KUKA KRL program: MyProgram_238().src

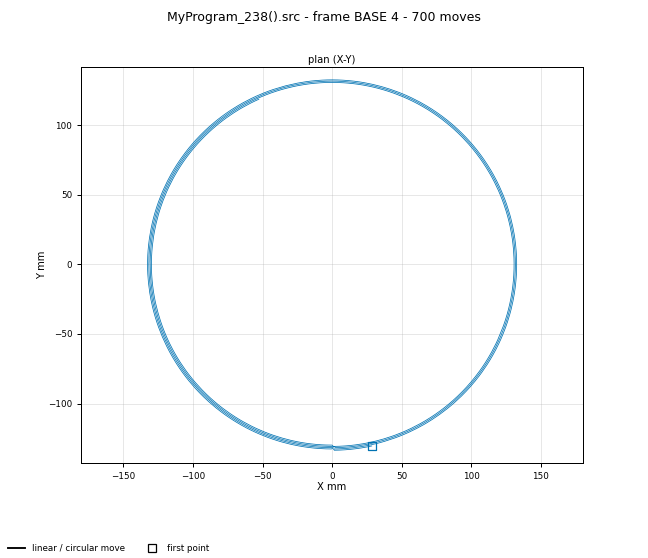
[picture p0: tool path of MyProgram_238().src in frame BASE 4, 700 of 700 moves have a stored position in this frame; points joined in program order, loops and branches not executed]
&ACCESS RVP
&REL 1
&PARAM TEMPLATE = C:\KRC\Roboter\Template\vorgabe
&PARAM EDITMASK = *
DEF MyProgram_238()
; ---- Setting reference (Base) ----
$BASE = BASE_DATA[4]

; --------------------------
; ---- Setting tool (TCP) ----
$TOOL = TOOL_DATA[3]
; --------------------------

$VEL.CP = VEL_APROX_PRINT
Startdeposition()
$VEL.CP = VEL_PRINT
LIN {X 28.5012,Y -130.5198,Z 160,A -79.1716,B 19.6548,C -0.4337,E1 19.6933,E2 527.426} C_DIS
LIN {X 25.4461,Y -131.1499,Z 160,A -80.7496,B 19.6549,C -0.4225,E1 19.6889,E2 529.0345} C_DIS
LIN {X 21.1826,Y -131.9073,Z 160,A -82.61,B 19.6549,C -0.4211,E1 19.6838,E2 530.8968} C_DIS
LIN {X 17.506,Y -132.4434,Z 160,A -84.1425,B 19.6549,C -0.4226,E1 19.6796,E2 532.4228} C_DIS
LIN {X 13.4148,Y -132.9217,Z 160,A -85.958,B 19.6549,C -0.4196,E1 19.6745,E2 534.2456} C_DIS
LIN {X 9.6729,Y -133.2447,Z 160,A -87.4931,B 19.6549,C -0.4221,E1 19.6703,E2 535.7723} C_DIS
LIN {X 5.6097,Y -133.4781,Z 160,A -89.2555,B 19.6549,C -0.4208,E1 19.6653,E2 537.5378} C_DIS
LIN {X 1.5658,Y -133.5878,Z 160,A -91.031,B 19.655,C -0.4187,E1 19.6604,E2 539.3193} C_DIS
LIN {X 1.5658,Y -133.5878,Z 160,A -91.031,B 19.655,C -0.4187,E1 19.6604,E2 539.3193} C_DIS
Enddeposition()
LIN {X 0.9434,Y -132.6616,Z 160,A -90.6102,B 18.4313,C -0.2923,E1 18.435,E2 539.1863} C_DIS
Startdeposition()
$VEL.CP = VEL_PRINT
LIN {X 3.7021,Y -132.6178,Z 160,A -88.9683,B 18.4311,C -0.31,E1 18.4397,E2 537.489} C_DIS
LIN {X 7.8936,Y -132.4346,Z 160,A -87.1638,B 18.4311,C -0.3103,E1 18.4447,E2 535.6844} C_DIS
LIN {X 11.5593,Y -132.1654,Z 160,A -85.513,B 18.431,C -0.3135,E1 18.4494,E2 534.0249} C_DIS
LIN {X 15.642,Y -131.744,Z 160,A -83.8719,B 18.431,C -0.3092,E1 18.4539,E2 532.3987} C_DIS
LIN {X 18.8772,Y -131.3195,Z 160,A -82.4668,B 18.431,C -0.3099,E1 18.4578,E2 530.9931} C_DIS
LIN {X 22.0168,Y -130.8298,Z 160,A -81.0377,B 18.431,C -0.3131,E1 18.4617,E2 529.556} C_DIS
LIN {X 27.2844,Y -129.8353,Z 160,A -78.6667,B 18.431,C -0.3171,E1 18.4682,E2 527.1765} C_DIS
LIN {X 31.009,Y -128.9944,Z 160,A -77.1259,B 18.431,C -0.3143,E1 18.4724,E2 525.6476} C_DIS
LIN {X 34.2185,Y -128.1803,Z 160,A -75.6772,B 18.431,C -0.3164,E1 18.4763,E2 524.1953} C_DIS
LIN {X 37.7119,Y -127.1971,Z 160,A -73.4165,B 18.4304,C -0.3458,E1 18.4826,E2 521.8475} C_DIS
LIN {X 42.8714,Y -125.5528,Z 160,A -71.8794,B 18.4309,C -0.3163,E1 18.4864,E2 520.4075} C_DIS
LIN {X 45.287,Y -124.7006,Z 160,A -70.7303,B 18.4309,C -0.3194,E1 18.4895,E2 519.2521} C_DIS
LIN {X 48.16,Y -123.6191,Z 160,A -69.3935,B 18.4309,C -0.3215,E1 18.493,E2 517.9126} C_DIS
LIN {X 51.5502,Y -122.245,Z 160,A -67.7549,B 18.4308,C -0.326,E1 18.4972,E2 516.2652} C_DIS
LIN {X 55.221,Y -120.6314,Z 160,A -65.2452,B 18.4302,C -0.36,E1 18.5038,E2 513.6571} C_DIS
LIN {X 60.6173,Y -118.0119,Z 160,A -63.7627,B 18.4309,C -0.3191,E1 18.5072,E2 512.3091} C_DIS
LIN {X 65.5426,Y -115.3507,Z 160,A -61.2737,B 18.4308,C -0.3259,E1 18.5133,E2 509.8088} C_DIS
LIN {X 68.1939,Y -113.8036,Z 160,A -59.6762,B 18.4306,C -0.3392,E1 18.5173,E2 508.1764} C_DIS
LIN {X 71.8599,Y -111.5251,Z 160,A -56.9687,B 18.4298,C -0.3771,E1 18.5239,E2 505.3617} C_DIS
LIN {X 77.3198,Y -107.8111,Z 160,A -55.0523,B 18.4305,C -0.3442,E1 18.528,E2 503.5582} C_DIS
LIN {X 82.5623,Y -103.851,Z 160,A -52.1665,B 18.4303,C -0.3519,E1 18.5344,E2 500.6629} C_DIS
LIN {X 85.006,Y -101.861,Z 160,A -50.9012,B 18.4303,C -0.3509,E1 18.5371,E2 499.4076} C_DIS
LIN {X 87.8381,Y -99.4285,Z 160,A -49.2007,B 18.4303,C -0.358,E1 18.5407,E2 497.6941} C_DIS
LIN {X 92.702,Y -94.91,Z 160,A -46.2129,B 18.43,C -0.3695,E1 18.5468,E2 494.6876} C_DIS
LIN {X 96.1781,Y -91.3865,Z 160,A -44.2202,B 18.43,C -0.3685,E1 18.5506,E2 492.7098} C_DIS
LIN {X 99.1469,Y -88.1567,Z 160,A -41.7561,B 18.4294,C -0.3968,E1 18.5554,E2 490.1723} C_DIS
LIN {X 102.5594,Y -84.1613,Z 160,A -40.2554,B 18.43,C -0.3705,E1 18.5579,E2 488.7637} C_DIS
LIN {X 105.6485,Y -80.2491,Z 160,A -37.9278,B 18.4297,C -0.3833,E1 18.5619,E2 486.4115} C_DIS
LIN {X 107.5535,Y -77.6779,Z 160,A -36.4631,B 18.4296,C -0.3903,E1 18.5643,E2 484.9345} C_DIS
LIN {X 111.3907,Y -72.0675,Z 160,A -33.8423,B 18.4296,C -0.3851,E1 18.5684,E2 482.3483} C_DIS
LIN {X 113.2763,Y -69.0665,Z 160,A -32.1365,B 18.4295,C -0.3965,E1 18.5709,E2 480.6186} C_DIS
LIN {X 115.4572,Y -65.3557,Z 160,A -30.138,B 18.4292,C -0.4075,E1 18.5737,E2 478.6} C_DIS
LIN {X 117.6562,Y -61.3044,Z 160,A -28.4402,B 18.4294,C -0.401,E1 18.5759,E2 476.9354} C_DIS
LIN {X 119.8553,Y -56.8847,Z 160,A -26.3011,B 18.4292,C -0.4074,E1 18.5785,E2 474.7922} C_DIS
LIN {X 121.3634,Y -53.5945,Z 160,A -24.7471,B 18.4292,C -0.4115,E1 18.5803,E2 473.2369} C_DIS
LIN {X 122.9377,Y -49.8746,Z 160,A -22.4308,B 18.4285,C -0.4406,E1 18.5828,E2 470.8472} C_DIS
LIN {X 124.6788,Y -45.3476,Z 160,A -21.1339,B 18.4291,C -0.4134,E1 18.584,E2 469.6456} C_DIS
LIN {X 126.0019,Y -41.5302,Z 160,A -19.0898,B 18.4287,C -0.4311,E1 18.5858,E2 467.5621} C_DIS
LIN {X 127.7829,Y -35.6739,Z 160,A -16.6066,B 18.4287,C -0.4324,E1 18.5878,E2 465.0946} C_DIS
LIN {X 128.6356,Y -32.4655,Z 160,A -15.1512,B 18.4286,C -0.4377,E1 18.5888,E2 463.6344} C_DIS
LIN {X 130.0281,Y -26.3408,Z 160,A -12.4494,B 18.4284,C -0.4456,E1 18.5904,E2 460.9299} C_DIS
LIN {X 130.9656,Y -21.2025,Z 160,A -10.1475,B 18.4282,C -0.4544,E1 18.5915,E2 458.6189} C_DIS
LIN {X 131.5378,Y -17.2906,Z 160,A -8.5274,B 18.4282,C -0.4561,E1 18.5922,E2 457.007} C_DIS
LIN {X 131.9613,Y -13.6979,Z 160,A -6.8849,B 18.4279,C -0.4643,E1 18.5927,E2 455.3523} C_DIS
LIN {X 132.3265,Y -9.5336,Z 160,A -5.2512,B 18.4279,C -0.4628,E1 18.593,E2 453.737} C_DIS
LIN {X 132.5387,Y -5.9326,Z 160,A -3.5264,B 18.4277,C -0.4746,E1 18.5933,E2 451.9894} C_DIS
LIN {X 132.6553,Y -1.9558,Z 160,A -1.9729,B 18.4277,C -0.473,E1 18.5933,E2 450.4536} C_DIS
LIN {X 132.6514,Y 2.1938,Z 160,A -0.1762,B 18.4276,C -0.4788,E1 18.5933,E2 448.6537} C_DIS
LIN {X 132.5359,Y 5.9882,Z 160,A 1.5365,B 18.4274,C -0.4869,E1 18.5931,E2 446.9298} C_DIS
LIN {X 132.3042,Y 9.8394,Z 160,A 3.135,B 18.4274,C -0.4893,E1 18.5928,E2 445.3372} C_DIS
LIN {X 131.9081,Y 14.1922,Z 160,A 4.9732,B 18.4272,C -0.493,E1 18.5923,E2 443.5024} C_DIS
LIN {X 131.3841,Y 18.4251,Z 160,A 6.8095,B 18.4271,C -0.4984,E1 18.5917,E2 441.6642} C_DIS
LIN {X 130.8489,Y 21.9018,Z 160,A 8.3213,B 18.427,C -0.5027,E1 18.591,E2 440.1513} C_DIS
LIN {X 129.8512,Y 27.2098,Z 160,A 11.4696,B 18.4258,C -0.5439,E1 18.5892,E2 436.8994} C_DIS
LIN {X 128.4247,Y 33.2964,Z 160,A 13.2373,B 18.4267,C -0.513,E1 18.5881,E2 435.2431} C_DIS
LIN {X 127.7028,Y 35.9602,Z 160,A 15.5458,B 18.4253,C -0.5632,E1 18.5862,E2 432.7954} C_DIS
LIN {X 125.4915,Y 43.0482,Z 160,A 17.4785,B 18.4265,C -0.5193,E1 18.5846,E2 431.0158} C_DIS
LIN {X 124.2159,Y 46.5992,Z 160,A 19.297,B 18.4262,C -0.5317,E1 18.5828,E2 429.1723} C_DIS
LIN {X 122.9726,Y 49.788,Z 160,A 20.729,B 18.4262,C -0.534,E1 18.5813,E2 427.7443} C_DIS
LIN {X 121.672,Y 52.8872,Z 160,A 22.1559,B 18.426,C -0.5371,E1 18.5798,E2 426.3188} C_DIS
LIN {X 120.3623,Y 55.8031,Z 160,A 23.5314,B 18.426,C -0.5407,E1 18.5782,E2 424.9423} C_DIS
LIN {X 118.2929,Y 60.0653,Z 160,A 25.2895,B 18.426,C -0.5344,E1 18.5761,E2 423.217} C_DIS
LIN {X 115.9637,Y 64.4518,Z 160,A 27.7485,B 18.4256,C -0.553,E1 18.5728,E2 420.7178} C_DIS
LIN {X 114.0137,Y 67.8413,Z 160,A 29.4654,B 18.4254,C -0.5586,E1 18.5703,E2 418.9957} C_DIS
LIN {X 111.6355,Y 71.6876,Z 160,A 31.3945,B 18.4253,C -0.5626,E1 18.5675,E2 417.0677} C_DIS
LIN {X 109.157,Y 75.4087,Z 160,A 33.3169,B 18.4251,C -0.567,E1 18.5644,E2 415.1445} C_DIS
LIN {X 106.6941,Y 78.8548,Z 160,A 35.137,B 18.4251,C -0.5711,E1 18.5614,E2 413.324} C_DIS
LIN {X 104.0345,Y 82.3317,Z 160,A 37.0312,B 18.4249,C -0.5757,E1 18.5582,E2 411.4277} C_DIS
LIN {X 101.3216,Y 85.6482,Z 160,A 38.8449,B 18.4249,C -0.5785,E1 18.555,E2 409.617} C_DIS
LIN {X 98.4834,Y 88.8971,Z 160,A 40.961,B 18.4244,C -0.5929,E1 18.551,E2 407.4687} C_DIS
LIN {X 96.0854,Y 91.4834,Z 160,A 42.2198,B 18.4246,C -0.5855,E1 18.5486,E2 406.2409} C_DIS
LIN {X 93.0242,Y 94.5944,Z 160,A 44.0784,B 18.4246,C -0.5883,E1 18.5449,E2 404.3842} C_DIS
LIN {X 89.9431,Y 97.5287,Z 160,A 45.9366,B 18.4244,C -0.5929,E1 18.5411,E2 402.5224} C_DIS
LIN {X 86.4794,Y 100.6125,Z 160,A 47.8719,B 18.4244,C -0.5941,E1 18.5371,E2 400.5941} C_DIS
LIN {X 83.3018,Y 103.2588,Z 160,A 49.8283,B 18.424,C -0.6042,E1 18.5328,E2 398.6161} C_DIS
LIN {X 78.6501,Y 106.8445,Z 160,A 52.182,B 18.424,C -0.6014,E1 18.5276,E2 396.2833} C_DIS
LIN {X 75.1653,Y 109.3241,Z 160,A 54.052,B 18.424,C -0.6054,E1 18.5233,E2 394.4097} C_DIS
LIN {X 71.3752,Y 111.8355,Z 160,A 55.9973,B 18.4239,C -0.6077,E1 18.5188,E2 392.466} C_DIS
LIN {X 67.7033,Y 114.0952,Z 160,A 57.9524,B 18.4237,C -0.6142,E1 18.5141,E2 390.4989} C_DIS
LIN {X 63.2262,Y 116.6368,Z 160,A 60.0969,B 18.4237,C -0.6142,E1 18.5089,E2 388.3634} C_DIS
LIN {X 59.9071,Y 118.3734,Z 160,A 61.5551,B 18.4238,C -0.61,E1 18.5053,E2 386.924} C_DIS
LIN {X 57.1185,Y 119.7436,Z 160,A 62.9333,B 18.4238,C -0.6131,E1 18.5018,E2 385.5412} C_DIS
LIN {X 53.9709,Y 121.195,Z 160,A 64.4173,B 18.4237,C -0.6143,E1 18.498,E2 384.0584} C_DIS
LIN {X 50.9379,Y 122.5007,Z 160,A 65.8351,B 18.4237,C -0.6156,E1 18.4944,E2 382.6415} C_DIS
LIN {X 47.9052,Y 123.7182,Z 160,A 67.2713,B 18.4236,C -0.618,E1 18.4906,E2 381.2021} C_DIS
LIN {X 44.4769,Y 124.9927,Z 160,A 68.7862,B 18.4236,C -0.6169,E1 18.4867,E2 379.6951} C_DIS
LIN {X 41.6904,Y 125.9486,Z 160,A 70.1214,B 18.4235,C -0.6205,E1 18.4831,E2 378.3522} C_DIS
LIN {X 35.2524,Y 127.9008,Z 160,A 73.0479,B 18.4234,C -0.6234,E1 18.4753,E2 375.4234} C_DIS
LIN {X 29.0695,Y 129.4461,Z 160,A 75.7411,B 18.4234,C -0.6228,E1 18.468,E2 372.7378} C_DIS
LIN {X 26.1718,Y 130.0624,Z 160,A 76.99,B 18.4234,C -0.6223,E1 18.4646,E2 371.4928} C_DIS
LIN {X 23.239,Y 130.6181,Z 160,A 78.3257,B 18.4234,C -0.6246,E1 18.4609,E2 370.1518} C_DIS
LIN {X 19.4787,Y 131.2335,Z 160,A 80.0834,B 18.4232,C -0.6295,E1 18.456,E2 368.3811} C_DIS
LIN {X 15.664,Y 131.7414,Z 160,A 81.6545,B 18.4232,C -0.6264,E1 18.4517,E2 366.8214} C_DIS
LIN {X 11.3785,Y 132.1807,Z 160,A 83.4808,B 18.4233,C -0.6254,E1 18.4466,E2 364.9998} C_DIS
LIN {X 7.9719,Y 132.4298,Z 160,A 84.9447,B 18.4233,C -0.6251,E1 18.4426,E2 363.5378} C_DIS
LIN {X 3.9853,Y 132.6099,Z 160,A 86.7034,B 18.4233,C -0.6264,E1 18.4376,E2 361.7757} C_DIS
LIN {X 0.1467,Y 132.6707,Z 160,A 88.3669,B 18.4233,C -0.6264,E1 18.433,E2 360.1123} C_DIS
LIN {X -3.5339,Y 132.6225,Z 160,A 89.9158,B 18.4233,C -0.6246,E1 18.4287,E2 358.569} C_DIS
LIN {X -7.0695,Y 132.4816,Z 160,A 91.4812,B 18.4233,C -0.6256,E1 18.4243,E2 357.0001} C_DIS
LIN {X -11.2701,Y 132.1899,Z 160,A 93.2615,B 18.4233,C -0.6235,E1 18.4194,E2 355.2254} C_DIS
LIN {X -15.1492,Y 131.8028,Z 160,A 95.0643,B 18.4233,C -0.6272,E1 18.4143,E2 353.4095} C_DIS
LIN {X -19.0348,Y 131.297,Z 160,A 96.7278,B 18.4233,C -0.6252,E1 18.4097,E2 351.7505} C_DIS
LIN {X -25.2457,Y 130.2455,Z 160,A 99.3709,B 18.4235,C -0.6204,E1 18.4025,E2 349.1186} C_DIS
LIN {X -33.5241,Y 128.3655,Z 160,A 102.9851,B 18.4237,C -0.6154,E1 18.3927,E2 345.5139} C_DIS
LIN {X -42.2415,Y 125.7651,Z 160,A 106.9794,B 18.4237,C -0.6137,E1 18.3821,E2 341.5156} C_DIS
LIN {X -45.5239,Y 124.6152,Z 160,A 108.64,B 18.4236,C -0.6177,E1 18.3776,E2 339.8375} C_DIS
LIN {X -49.4917,Y 123.092,Z 160,A 111.0393,B 18.423,C -0.6361,E1 18.3712,E2 337.3724} C_DIS
LIN {X -54.3882,Y 121.0084,Z 160,A 112.6667,B 18.4239,C -0.6084,E1 18.3673,E2 335.8277} C_DIS
LIN {X -58.0987,Y 119.2729,Z 160,A 115.4054,B 18.4228,C -0.6412,E1 18.3602,E2 332.9746} C_DIS
LIN {X -64.1253,Y 116.1445,Z 160,A 117.4669,B 18.424,C -0.6047,E1 18.3553,E2 331.0211} C_DIS
LIN {X -68.0267,Y 113.9032,Z 160,A 119.4005,B 18.4241,C -0.6011,E1 18.3507,E2 329.0909} C_DIS
LIN {X -72.5443,Y 111.0812,Z 160,A 121.5933,B 18.4244,C -0.5931,E1 18.3456,E2 326.9137} C_DIS
LIN {X -75.4962,Y 109.0963,Z 160,A 123.622,B 18.4239,C -0.608,E1 18.3408,E2 324.8281} C_DIS
LIN {X -78.7284,Y 106.7869,Z 160,A 124.88,B 18.4245,C -0.5882,E1 18.338,E2 323.6268} C_DIS
LIN {X -81.7101,Y 104.5233,Z 160,A 126.63,B 18.4245,C -0.5897,E1 18.3341,E2 321.863} C_DIS
LIN {X -84.669,Y 102.1407,Z 160,A 128.2475,B 18.4245,C -0.5855,E1 18.3307,E2 320.2504} C_DIS
LIN {X -88.3447,Y 98.9789,Z 160,A 130.3934,B 18.4247,C -0.5829,E1 18.3261,E2 318.1011} C_DIS
LIN {X -91.5366,Y 96.0346,Z 160,A 132.7692,B 18.4242,C -0.5966,E1 18.3212,E2 315.668} C_DIS
LIN {X -94.939,Y 92.6728,Z 160,A 134.7487,B 18.4245,C -0.5887,E1 18.3174,E2 313.7016} C_DIS
LIN {X -97.8577,Y 89.5852,Z 160,A 135.9447,B 18.4253,C -0.5617,E1 18.3153,E2 312.5844} C_DIS
LIN {X -99.9652,Y 87.2269,Z 160,A 137.5668,B 18.4251,C -0.5674,E1 18.3122,E2 310.9337} C_DIS
LIN {X -102.7832,Y 83.8879,Z 160,A 139.4582,B 18.4253,C -0.5629,E1 18.3088,E2 309.0446} C_DIS
LIN {X -105.4862,Y 80.4628,Z 160,A 141.5221,B 18.4253,C -0.5645,E1 18.3053,E2 306.962} C_DIS
LIN {X -108.8277,Y 75.8823,Z 160,A 144.3991,B 18.425,C -0.5732,E1 18.3006,E2 304.0373} C_DIS
LIN {X -111.6585,Y 71.6517,Z 160,A 146.404,B 18.4253,C -0.5604,E1 18.2976,E2 302.0589} C_DIS
LIN {X -113.7843,Y 68.2263,Z 160,A 147.6631,B 18.426,C -0.5387,E1 18.2958,E2 300.8599} C_DIS
LIN {X -115.5744,Y 65.1471,Z 160,A 149.36,B 18.426,C -0.54,E1 18.2935,E2 299.1464} C_DIS
LIN {X -118.3896,Y 59.8754,Z 160,A 152.1829,B 18.4259,C -0.5413,E1 18.2898,E2 296.2985} C_DIS
LIN {X -119.864,Y 56.8665,Z 160,A 153.2968,B 18.4263,C -0.5255,E1 18.2885,E2 295.2266} C_DIS
LIN {X -121.1397,Y 54.0946,Z 160,A 154.6403,B 18.4264,C -0.5226,E1 18.287,E2 293.882} C_DIS
LIN {X -122.66,Y 50.5566,Z 160,A 156.3085,B 18.4265,C -0.5179,E1 18.2851,E2 292.2158} C_DIS
LIN {X -123.7991,Y 47.697,Z 160,A 157.6411,B 18.4266,C -0.5141,E1 18.2838,E2 290.8847} C_DIS
LIN {X -124.8407,Y 44.8986,Z 160,A 158.9985,B 18.4266,C -0.5126,E1 18.2825,E2 289.5212} C_DIS
LIN {X -126.1094,Y 41.2074,Z 160,A 160.8063,B 18.4267,C -0.5118,E1 18.2809,E2 287.7015} C_DIS
LIN {X -127.3043,Y 37.3459,Z 160,A 162.4601,B 18.4269,C -0.5034,E1 18.2796,E2 286.0612} C_DIS
LIN {X -128.3322,Y 33.6489,Z 160,A 164.0639,B 18.4271,C -0.4965,E1 18.2784,E2 284.4664} C_DIS
LIN {X -129.1541,Y 30.3465,Z 160,A 165.7119,B 18.4271,C -0.4982,E1 18.2773,E2 282.7994} C_DIS
LIN {X -130.078,Y 26.0955,Z 160,A 167.292,B 18.4275,C -0.4821,E1 18.2764,E2 281.2576} C_DIS
LIN {X -131.3056,Y 18.9746,Z 160,A 170.3774,B 18.4278,C -0.4712,E1 18.275,E2 278.1814} C_DIS
LIN {X -131.9478,Y 13.8234,Z 160,A 173.0684,B 18.4275,C -0.4798,E1 18.2741,E2 275.4402} C_DIS
LIN {X -132.2894,Y 10.0418,Z 160,A 174.6013,B 18.4278,C -0.471,E1 18.2737,E2 273.9227} C_DIS
LIN {X -132.5134,Y 6.4374,Z 160,A 176.1557,B 18.4278,C -0.4659,E1 18.2735,E2 272.3712} C_DIS
LIN {X -132.6695,Y 0.5426,Z 160,A 178.9475,B 18.4278,C -0.4666,E1 18.2734,E2 269.5537} C_DIS
LIN {X -132.6236,Y -3.4935,Z 160,A -179.5425,B 18.4282,C -0.453,E1 18.2734,E2 268.0742} C_DIS
LIN {X -132.4931,Y -6.8404,Z 160,A -178.0813,B 18.4282,C -0.4491,E1 18.2736,E2 266.6133} C_DIS
LIN {X -132.0412,Y -12.8967,Z 160,A -175.528,B 18.4285,C -0.4385,E1 18.2742,E2 264.072} C_DIS
LIN {X -131.0844,Y -20.4463,Z 160,A -172.2438,B 18.4288,C -0.4284,E1 18.2754,E2 260.7928} C_DIS
LIN {X -130.136,Y -25.8105,Z 160,A -169.4662,B 18.4286,C -0.4361,E1 18.2769,E2 257.9675} C_DIS
LIN {X -129.0551,Y -30.7573,Z 160,A -167.5305,B 18.4289,C -0.4208,E1 18.278,E2 256.0647} C_DIS
LIN {X -128.2042,Y -34.1288,Z 160,A -166.0109,B 18.429,C -0.4169,E1 18.2791,E2 254.5449} C_DIS
LIN {X -127.1442,Y -37.8927,Z 160,A -164.2814,B 18.429,C -0.4134,E1 18.2804,E2 252.8127} C_DIS
LIN {X -125.9564,Y -41.6669,Z 160,A -162.624,B 18.4292,C -0.4066,E1 18.2819,E2 251.1635} C_DIS
LIN {X -124.7652,Y -45.1079,Z 160,A -161.0348,B 18.4293,C -0.4027,E1 18.2833,E2 249.5742} C_DIS
LIN {X -123.0247,Y -49.6588,Z 160,A -159.2636,B 18.4297,C -0.385,E1 18.2851,E2 247.8454} C_DIS
LIN {X -121.9684,Y -52.2016,Z 160,A -157.6531,B 18.4295,C -0.3965,E1 18.2869,E2 246.1858} C_DIS
LIN {X -118.8589,Y -58.9378,Z 160,A -154.4318,B 18.4296,C -0.3883,E1 18.2907,E2 242.966} C_DIS
LIN {X -116.7092,Y -63.0924,Z 160,A -152.3373,B 18.4296,C -0.3855,E1 18.2934,E2 240.8648} C_DIS
LIN {X -114.2671,Y -67.4141,Z 160,A -150.1858,B 18.4298,C -0.3802,E1 18.2964,E2 238.7145} C_DIS
LIN {X -111.9536,Y -71.1907,Z 160,A -147.8094,B 18.4295,C -0.392,E1 18.3001,E2 236.2837} C_DIS
LIN {X -109.4746,Y -74.946,Z 160,A -146.5251,B 18.4301,C -0.3635,E1 18.302,E2 235.0811} C_DIS
LIN {X -107.6334,Y -77.5676,Z 160,A -144.8757,B 18.43,C -0.3697,E1 18.3047,E2 233.4009} C_DIS
LIN {X -104.996,Y -81.1015,Z 160,A -142.763,B 18.43,C -0.3727,E1 18.3083,E2 231.2645} C_DIS
LIN {X -102.8864,Y -83.7617,Z 160,A -141.4959,B 18.4301,C -0.3621,E1 18.3105,E2 230.0228} C_DIS
LIN {X -98.3138,Y -89.084,Z 160,A -138.4797,B 18.4303,C -0.3548,E1 18.316,E2 227.0107} C_DIS
LIN {X -95.4309,Y -92.1658,Z 160,A -136.6227,B 18.4303,C -0.3522,E1 18.3196,E2 225.1508} C_DIS
LIN {X -92.2744,Y -95.3257,Z 160,A -134.539,B 18.4303,C -0.3539,E1 18.3238,E2 223.0496} C_DIS
LIN {X -88.7175,Y -98.645,Z 160,A -132.5605,B 18.4304,C -0.3453,E1 18.3278,E2 221.0872} C_DIS
LIN {X -83.383,Y -103.1933,Z 160,A -129.5421,B 18.4306,C -0.3393,E1 18.3343,E2 218.0718} C_DIS
LIN {X -79.9809,Y -105.8519,Z 160,A -127.6742,B 18.4306,C -0.3361,E1 18.3384,E2 216.2044} C_DIS
LIN {X -76.4095,Y -108.4581,Z 160,A -125.7745,B 18.4306,C -0.3326,E1 18.3427,E2 214.3067} C_DIS
LIN {X -72.8618,Y -110.8726,Z 160,A -123.8912,B 18.4307,C -0.3307,E1 18.3471,E2 212.4205} C_DIS
LIN {X -69.241,Y -113.1692,Z 160,A -121.9537,B 18.4307,C -0.3312,E1 18.3517,E2 210.4731} C_DIS
LIN {X -65.2017,Y -115.5437,Z 160,A -120.0005,B 18.4307,C -0.3257,E1 18.3564,E2 208.5291} C_DIS
LIN {X -61.4859,Y -117.5609,Z 160,A -118.2437,B 18.4309,C -0.3208,E1 18.3607,E2 206.7812} C_DIS
LIN {X -58.478,Y -119.0858,Z 160,A -116.8046,B 18.4309,C -0.3184,E1 18.3643,E2 205.3444} C_DIS
LIN {X -55.5076,Y -120.4989,Z 160,A -115.3716,B 18.4309,C -0.3172,E1 18.368,E2 203.9101} C_DIS
LIN {X -52.5429,Y -121.8208,Z 160,A -113.9582,B 18.4309,C -0.3161,E1 18.3716,E2 202.4955} C_DIS
LIN {X -49.3738,Y -123.1395,Z 160,A -112.5064,B 18.4309,C -0.3134,E1 18.3753,E2 201.0476} C_DIS
LIN {X -46.4199,Y -124.283,Z 160,A -111.1267,B 18.431,C -0.3126,E1 18.3789,E2 199.6665} C_DIS
LIN {X -43.0906,Y -125.4768,Z 160,A -109.0927,B 18.4307,C -0.3305,E1 18.3845,E2 197.5706} C_DIS
LIN {X -39.114,Y -126.7725,Z 160,A -107.9733,B 18.4312,C -0.3031,E1 18.3872,E2 196.5352} C_DIS
LIN {X -36.0543,Y -127.6765,Z 160,A -105.6146,B 18.4306,C -0.3394,E1 18.3939,E2 194.056} C_DIS
LIN {X -30.5064,Y -129.1155,Z 160,A -103.9633,B 18.4311,C -0.3065,E1 18.3981,E2 192.5059} C_DIS
LIN {X -28.0053,Y -129.6797,Z 160,A -102.7826,B 18.4311,C -0.3088,E1 18.4013,E2 191.3159} C_DIS
LIN {X -24.3122,Y -130.424,Z 160,A -101.0439,B 18.4311,C -0.3124,E1 18.4061,E2 189.5633} C_DIS
LIN {X -20.3202,Y -131.1039,Z 160,A -99.4397,B 18.4311,C -0.3063,E1 18.4105,E2 187.9762} C_DIS
LIN {X -16.9585,Y -131.5813,Z 160,A -97.8589,B 18.4311,C -0.3103,E1 18.4149,E2 186.3811} C_DIS
LIN {X -12.7411,Y -132.0562,Z 160,A -96.0917,B 18.4311,C -0.3075,E1 18.4198,E2 184.6213} C_DIS
LIN {X -8.616,Y -132.3901,Z 160,A -94.2446,B 18.4311,C -0.3097,E1 18.425,E2 182.7662} C_DIS
LIN {X -4.3375,Y -132.6002,Z 160,A -92.3692,B 18.4311,C -0.3108,E1 18.4302,E2 180.8869} C_DIS
LIN {X -0.4314,Y -132.6692,Z 160,A -90.6709,B 18.4311,C -0.3115,E1 18.435,E2 179.1863} C_DIS
LIN {X -0.4314,Y -132.6692,Z 160,A -90.6709,B 18.4311,C -0.3115,E1 18.435,E2 179.1863} C_DIS
Enddeposition()
LIN {X 0.9315,Y -131.7392,Z 160,A -89.7694,B 16.8849,C -0.1477,E1 16.8882,E2 178.7145} C_DIS
Startdeposition()
$VEL.CP = VEL_PRINT
LIN {X -3.0382,Y -131.71,Z 160,A -92.225,B 16.8851,C -0.1219,E1 16.8811,E2 181.259} C_DIS
LIN {X -6.8947,Y -131.5633,Z 160,A -93.7694,B 16.8851,C -0.1265,E1 16.8768,E2 182.788} C_DIS
LIN {X -10.6205,Y -131.3155,Z 160,A -95.4821,B 16.8851,C -0.1236,E1 16.872,E2 184.512} C_DIS
LIN {X -14.1826,Y -130.9778,Z 160,A -96.9934,B 16.8851,C -0.1253,E1 16.8678,E2 186.0184} C_DIS
LIN {X -17.6017,Y -130.5632,Z 160,A -98.6003,B 16.8851,C -0.1219,E1 16.8633,E2 187.6388} C_DIS
LIN {X -21.7395,Y -129.9373,Z 160,A -100.305,B 16.8851,C -0.1264,E1 16.8587,E2 189.3302} C_DIS
LIN {X -25.5308,Y -129.248,Z 160,A -102.1164,B 16.8851,C -0.1225,E1 16.8537,E2 191.1583} C_DIS
LIN {X -29.4249,Y -128.4152,Z 160,A -104.4591,B 16.8852,C -0.1027,E1 16.8471,E2 193.5737} C_DIS
LIN {X -34.8461,Y -127.053,Z 160,A -106.0777,B 16.885,C -0.1316,E1 16.843,E2 195.0962} C_DIS
LIN {X -41.0436,Y -125.1881,Z 160,A -108.8793,B 16.885,C -0.1341,E1 16.8355,E2 197.8966} C_DIS
LIN {X -43.5556,Y -124.3356,Z 160,A -110.2625,B 16.885,C -0.1274,E1 16.8318,E2 199.3071} C_DIS
LIN {X -47.5527,Y -122.8618,Z 160,A -111.9804,B 16.885,C -0.1336,E1 16.8273,E2 201.0088} C_DIS
LIN {X -50.705,Y -121.5946,Z 160,A -113.4476,B 16.885,C -0.1355,E1 16.8235,E2 202.4747} C_DIS
LIN {X -53.8598,Y -120.2304,Z 160,A -114.9612,B 16.885,C -0.1365,E1 16.8197,E2 203.9905} C_DIS
LIN {X -56.844,Y -118.8486,Z 160,A -116.4209,B 16.885,C -0.1371,E1 16.816,E2 205.4535} C_DIS
LIN {X -60.1312,Y -117.2204,Z 160,A -118.1103,B 16.885,C -0.136,E1 16.8117,E2 207.1537} C_DIS
LIN {X -64.0985,Y -115.1009,Z 160,A -120.0509,B 16.885,C -0.139,E1 16.807,E2 209.0922} C_DIS
LIN {X -67.656,Y -113.0463,Z 160,A -121.9016,B 16.885,C -0.1395,E1 16.8025,E2 210.95} C_DIS
LIN {X -70.8955,Y -111.0432,Z 160,A -123.5301,B 16.885,C -0.1429,E1 16.7987,E2 212.5746} C_DIS
LIN {X -74.7646,Y -108.4761,Z 160,A -125.566,B 16.885,C -0.1455,E1 16.7939,E2 214.6119} C_DIS
LIN {X -78.3556,Y -105.9117,Z 160,A -127.5146,B 16.885,C -0.1477,E1 16.7895,E2 216.5632} C_DIS
LIN {X -81.896,Y -103.198,Z 160,A -129.775,B 16.885,C -0.1408,E1 16.7845,E2 218.8605} C_DIS
LIN {X -84.9102,Y -100.7317,Z 160,A -131.3333,B 16.8849,C -0.1483,E1 16.7812,E2 220.402} C_DIS
LIN {X -87.3568,Y -98.6182,Z 160,A -132.274,B 16.8847,C -0.166,E1 16.7793,E2 221.2869} C_DIS
LIN {X -89.7338,Y -96.4602,Z 160,A -133.9635,B 16.8848,C -0.1592,E1 16.7758,E2 223.0104} C_DIS
LIN {X -92.2738,Y -94.0334,Z 160,A -135.486,B 16.8848,C -0.1625,E1 16.7727,E2 224.5314} C_DIS
LIN {X -95.4387,Y -90.82,Z 160,A -137.4686,B 16.8848,C -0.1659,E1 16.7689,E2 226.5153} C_DIS
LIN {X -101.1001,Y -84.4724,Z 160,A -141.5785,B 16.8848,C -0.161,E1 16.7613,E2 230.6708} C_DIS
LIN {X -103.7084,Y -81.2485,Z 160,A -142.7614,B 16.8845,C -0.1849,E1 16.7594,E2 231.7793} C_DIS
LIN {X -105.5916,Y -78.7855,Z 160,A -144.3743,B 16.8846,C -0.1796,E1 16.7566,E2 233.4225} C_DIS
LIN {X -108.2915,Y -75.0317,Z 160,A -146.6934,B 16.8846,C -0.1747,E1 16.7528,E2 235.7761} C_DIS
LIN {X -110.3395,Y -71.9848,Z 160,A -148.152,B 16.8846,C -0.183,E1 16.7506,E2 237.2171} C_DIS
LIN {X -112.313,Y -68.866,Z 160,A -149.6388,B 16.8845,C -0.1908,E1 16.7484,E2 238.6887} C_DIS
LIN {X -114.3681,Y -65.3965,Z 160,A -151.1783,B 16.8844,C -0.2021,E1 16.7463,E2 240.2013} C_DIS
LIN {X -115.8732,Y -62.692,Z 160,A -152.7766,B 16.8844,C -0.1976,E1 16.7441,E2 241.828} C_DIS
LIN {X -117.8994,Y -58.79,Z 160,A -155.4422,B 16.8846,C -0.1792,E1 16.7407,E2 244.5795} C_DIS
LIN {X -120.4988,Y -53.2598,Z 160,A -157.3043,B 16.8842,C -0.2112,E1 16.7387,E2 246.3463} C_DIS
LIN {X -121.7958,Y -50.2233,Z 160,A -159.0598,B 16.8843,C -0.2052,E1 16.7367,E2 248.1376} C_DIS
LIN {X -123.1112,Y -46.9087,Z 160,A -160.2287,B 16.8841,C -0.2215,E1 16.7356,E2 249.2601} C_DIS
LIN {X -124.3319,Y -43.5662,Z 160,A -161.8843,B 16.8841,C -0.2225,E1 16.734,E2 250.9267} C_DIS
LIN {X -125.4522,Y -40.2248,Z 160,A -163.3645,B 16.8841,C -0.2285,E1 16.7328,E2 252.399} C_DIS
LIN {X -126.4668,Y -36.9112,Z 160,A -164.8919,B 16.884,C -0.2322,E1 16.7315,E2 253.927} C_DIS
LIN {X -127.3997,Y -33.5523,Z 160,A -166.3899,B 16.884,C -0.2372,E1 16.7304,E2 255.4211} C_DIS
LIN {X -128.1989,Y -30.3579,Z 160,A -168.293,B 16.884,C -0.2268,E1 16.7292,E2 257.3775} C_DIS
LIN {X -129.0218,Y -26.6426,Z 160,A -169.8083,B 16.884,C -0.2361,E1 16.7283,E2 258.8745} C_DIS
LIN {X -130.0114,Y -21.2954,Z 160,A -171.9095,B 16.8837,C -0.2513,E1 16.7273,E2 260.942} C_DIS
LIN {X -130.8597,Y -15.238,Z 160,A -174.5632,B 16.8836,C -0.2595,E1 16.7263,E2 263.5916} C_DIS
LIN {X -131.4914,Y -8.1463,Z 160,A -177.7187,B 16.8835,C -0.267,E1 16.7256,E2 266.7501} C_DIS
LIN {X -131.6699,Y -4.4547,Z 160,A -179.9048,B 16.8837,C -0.2541,E1 16.7254,E2 269.0015} C_DIS
LIN {X -131.7465,Y 0.0689,Z 160,A 177.9636,B 16.8837,C -0.2551,E1 16.7254,E2 271.1493} C_DIS
LIN {X -131.6448,Y 5.0991,Z 160,A 176.6116,B 16.8832,C -0.2875,E1 16.7254,E2 272.4012} C_DIS
LIN {X -131.496,Y 8.0712,Z 160,A 174.667,B 16.8834,C -0.2715,E1 16.7258,E2 274.4197} C_DIS
LIN {X -131.1806,Y 12.1723,Z 160,A 173.0412,B 16.8832,C -0.2819,E1 16.7262,E2 276.0241} C_DIS
LIN {X -130.6121,Y 17.2284,Z 160,A 171.1286,B 16.883,C -0.298,E1 16.7268,E2 277.8987} C_DIS
LIN {X -130.1567,Y 20.3862,Z 160,A 169.1897,B 16.8832,C -0.2852,E1 16.7277,E2 279.8996} C_DIS
LIN {X -129.431,Y 24.5751,Z 160,A 167.811,B 16.8829,C -0.3053,E1 16.7284,E2 281.2213} C_DIS
LIN {X -128.4922,Y 29.088,Z 160,A 166.0368,B 16.8826,C -0.3185,E1 16.7294,E2 282.9657} C_DIS
LIN {X -127.7864,Y 32.0475,Z 160,A 164.3999,B 16.8827,C -0.3127,E1 16.7305,E2 284.6374} C_DIS
LIN {X -126.8029,Y 35.7402,Z 160,A 162.8097,B 16.8826,C -0.3199,E1 16.7316,E2 286.2168} C_DIS
LIN {X -125.7474,Y 39.2997,Z 160,A 160.9447,B 16.8826,C -0.3169,E1 16.7332,E2 288.1087} C_DIS
LIN {X -124.4121,Y 43.3349,Z 160,A 159.2749,B 16.8824,C -0.3279,E1 16.7347,E2 289.7551} C_DIS
LIN {X -123.0528,Y 47.0614,Z 160,A 157.3226,B 16.8824,C -0.3259,E1 16.7366,E2 291.7312} C_DIS
LIN {X -121.3612,Y 51.2638,Z 160,A 155.5811,B 16.8822,C -0.3387,E1 16.7384,E2 293.4434} C_DIS
LIN {X -120.072,Y 54.214,Z 160,A 154.1471,B 16.8822,C -0.3416,E1 16.74,E2 294.8794} C_DIS
LIN {X -118.5345,Y 57.5014,Z 160,A 152.3995,B 16.8822,C -0.3408,E1 16.7422,E2 296.6444} C_DIS
LIN {X -115.7538,Y 62.9114,Z 160,A 149.8111,B 16.882,C -0.3499,E1 16.7455,E2 299.2224} C_DIS
LIN {X -113.6314,Y 66.6682,Z 160,A 147.7274,B 16.882,C -0.3485,E1 16.7485,E2 301.3274} C_DIS
LIN {X -111.5856,Y 70.0394,Z 160,A 146.175,B 16.8818,C -0.3581,E1 16.7507,E2 302.8587} C_DIS
LIN {X -108.4005,Y 74.8747,Z 160,A 143.6484,B 16.8818,C -0.3645,E1 16.7546,E2 305.3828} C_DIS
LIN {X -105.8287,Y 78.4669,Z 160,A 141.6105,B 16.8817,C -0.3657,E1 16.758,E2 307.4316} C_DIS
LIN {X -103.5918,Y 81.397,Z 160,A 140.0962,B 16.8815,C -0.3725,E1 16.7606,E2 308.9333} C_DIS
LIN {X -100.6981,Y 84.9515,Z 160,A 138.0719,B 16.8815,C -0.3764,E1 16.7642,E2 310.9586} C_DIS
LIN {X -97.8202,Y 88.25,Z 160,A 136.2147,B 16.8813,C -0.3823,E1 16.7676,E2 312.8078} C_DIS
LIN {X -94.2823,Y 92.0201,Z 160,A 133.6414,B 16.8814,C -0.3773,E1 16.7726,E2 315.4157} C_DIS
LIN {X -91.8305,Y 94.4668,Z 160,A 132.3682,B 16.8812,C -0.388,E1 16.7751,E2 316.6601} C_DIS
LIN {X -88.6508,Y 97.4567,Z 160,A 130.5101,B 16.8811,C -0.3934,E1 16.7789,E2 318.5112} C_DIS
LIN {X -85.2619,Y 100.4348,Z 160,A 128.64,B 16.8809,C -0.4004,E1 16.7828,E2 320.3681} C_DIS
LIN {X -82.5887,Y 102.6443,Z 160,A 127.2511,B 16.8808,C -0.4073,E1 16.7858,E2 321.7413} C_DIS
LIN {X -80.2562,Y 104.4785,Z 160,A 125.6557,B 16.8809,C -0.4001,E1 16.7894,E2 323.3705} C_DIS
LIN {X -74.4713,Y 108.6774,Z 160,A 122.6294,B 16.8807,C -0.4085,E1 16.7962,E2 326.3837} C_DIS
LIN {X -69.9785,Y 111.624,Z 160,A 120.3834,B 16.8806,C -0.4156,E1 16.8015,E2 328.6166} C_DIS
LIN {X -67.1733,Y 113.334,Z 160,A 118.7553,B 16.8806,C -0.4115,E1 16.8054,E2 330.2662} C_DIS
LIN {X -63.2609,Y 115.5632,Z 160,A 115.9747,B 16.8812,C -0.3884,E1 16.8125,E2 333.1391} C_DIS
LIN {X -57.5998,Y 118.4866,Z 160,A 114.0906,B 16.8804,C -0.4209,E1 16.8169,E2 334.9185} C_DIS
LIN {X -50.2016,Y 121.8048,Z 160,A 110.6218,B 16.8803,C -0.4274,E1 16.8257,E2 338.3773} C_DIS
LIN {X -47.5351,Y 122.8686,Z 160,A 109.2883,B 16.8803,C -0.4262,E1 16.8292,E2 339.7195} C_DIS
LIN {X -43.4999,Y 124.3549,Z 160,A 107.311,B 16.8803,C -0.4248,E1 16.8344,E2 341.7074} C_DIS
LIN {X -36.7765,Y 126.5062,Z 160,A 104.4241,B 16.8801,C -0.434,E1 16.8421,E2 344.5704} C_DIS
LIN {X -33.9477,Y 127.2943,Z 160,A 102.7156,B 16.8804,C -0.421,E1 16.8468,E2 346.3279} C_DIS
LIN {X -30.5025,Y 128.1638,Z 160,A 101.2007,B 16.8804,C -0.4232,E1 16.8509,E2 347.8381} C_DIS
LIN {X -27.1088,Y 128.926,Z 160,A 100.0881,B 16.88,C -0.4376,E1 16.8538,E2 348.9033} C_DIS
LIN {X -20.8348,Y 130.0873,Z 160,A 97.1317,B 16.8801,C -0.4333,E1 16.862,E2 351.8789} C_DIS
LIN {X -16.8688,Y 130.6592,Z 160,A 95.4098,B 16.8801,C -0.4349,E1 16.8668,E2 353.5972} C_DIS
LIN {X -12.6593,Y 131.1338,Z 160,A 93.6114,B 16.8801,C -0.4372,E1 16.8717,E2 355.3893} C_DIS
LIN {X -8.6865,Y 131.4581,Z 160,A 91.7936,B 16.8801,C -0.435,E1 16.8768,E2 357.216} C_DIS
LIN {X -4.831,Y 131.6553,Z 160,A 90.1647,B 16.8801,C -0.4371,E1 16.8813,E2 358.8381} C_DIS
LIN {X -0.6416,Y 131.7421,Z 160,A 88.3998,B 16.88,C -0.4393,E1 16.8863,E2 360.5954} C_DIS
LIN {X 3.3295,Y 131.7019,Z 160,A 86.6081,B 16.88,C -0.4372,E1 16.8913,E2 362.3938} C_DIS
LIN {X 7.1481,Y 131.5505,Z 160,A 84.8875,B 16.88,C -0.4352,E1 16.8961,E2 364.1205} C_DIS
LIN {X 11.1408,Y 131.2716,Z 160,A 83.2475,B 16.88,C -0.4384,E1 16.9006,E2 365.7482} C_DIS
LIN {X 15.3251,Y 130.8493,Z 160,A 81.4139,B 16.88,C -0.4378,E1 16.9057,E2 367.5817} C_DIS
LIN {X 19.0683,Y 130.3569,Z 160,A 79.8632,B 16.88,C -0.4405,E1 16.91,E2 369.1213} C_DIS
LIN {X 21.8465,Y 129.9195,Z 160,A 78.5524,B 16.88,C -0.437,E1 16.9136,E2 370.442} C_DIS
LIN {X 26.0802,Y 129.1362,Z 160,A 76.6905,B 16.88,C -0.4365,E1 16.9187,E2 372.3023} C_DIS
LIN {X 31.1084,Y 128.018,Z 160,A 74.4447,B 16.88,C -0.435,E1 16.9248,E2 374.5484} C_DIS
LIN {X 37.9546,Y 126.1591,Z 160,A 71.4787,B 16.88,C -0.4369,E1 16.9328,E2 377.5001} C_DIS
LIN {X 42.0211,Y 124.8626,Z 160,A 69.5937,B 16.8801,C -0.4344,E1 16.9378,E2 379.3885} C_DIS
LIN {X 44.8797,Y 123.8633,Z 160,A 68.2137,B 16.8801,C -0.431,E1 16.9414,E2 380.7758} C_DIS
LIN {X 48.145,Y 122.6316,Z 160,A 66.7314,B 16.8801,C -0.4307,E1 16.9453,E2 382.254} C_DIS
LIN {X 51.1702,Y 121.4003,Z 160,A 65.3393,B 16.8802,C -0.4302,E1 16.9489,E2 383.6429} C_DIS
LIN {X 53.9426,Y 120.1934,Z 160,A 63.9864,B 16.8802,C -0.4274,E1 16.9523,E2 385.0004} C_DIS
LIN {X 57.3139,Y 118.6241,Z 160,A 62.3561,B 16.8803,C -0.425,E1 16.9565,E2 386.6324} C_DIS
LIN {X 60.6714,Y 116.9428,Z 160,A 60.7317,B 16.8803,C -0.4232,E1 16.9605,E2 388.2562} C_DIS
LIN {X 64.1821,Y 115.0546,Z 160,A 58.9079,B 16.8805,C -0.4176,E1 16.965,E2 390.091} C_DIS
LIN {X 68.7217,Y 112.4016,Z 160,A 56.9995,B 16.8803,C -0.4278,E1 16.9695,E2 391.9555} C_DIS
LIN {X 71.1067,Y 110.908,Z 160,A 55.4394,B 16.8806,C -0.4138,E1 16.9733,E2 393.5555} C_DIS
LIN {X 74.7734,Y 108.4701,Z 160,A 53.5369,B 16.8806,C -0.4112,E1 16.9777,E2 395.4573} C_DIS
LIN {X 78.1629,Y 106.0535,Z 160,A 51.7462,B 16.8807,C -0.4088,E1 16.9817,E2 397.2463} C_DIS
LIN {X 81.4709,Y 103.5337,Z 160,A 49.8236,B 16.8809,C -0.4015,E1 16.986,E2 399.1832} C_DIS
LIN {X 84.9386,Y 100.7089,Z 160,A 47.997,B 16.8809,C -0.4021,E1 16.9899,E2 400.9968} C_DIS
LIN {X 88.2572,Y 97.8138,Z 160,A 46.0635,B 16.8809,C -0.3978,E1 16.9939,E2 402.9335} C_DIS
LIN {X 91.4799,Y 94.8062,Z 160,A 44.1817,B 16.881,C -0.3952,E1 16.9977,E2 404.8122} C_DIS
LIN {X 94.5571,Y 91.7371,Z 160,A 42.2738,B 16.8811,C -0.3906,E1 17.0015,E2 406.7234} C_DIS
LIN {X 98.2468,Y 87.7743,Z 160,A 40.0421,B 16.8811,C -0.3899,E1 17.0057,E2 408.9422} C_DIS
LIN {X 100.9116,Y 84.6971,Z 160,A 38.223,B 16.8813,C -0.3842,E1 17.009,E2 410.7683} C_DIS
LIN {X 103.6821,Y 81.2821,Z 160,A 36.3153,B 16.8813,C -0.3799,E1 17.0123,E2 412.6768} C_DIS
LIN {X 106.3849,Y 77.7118,Z 160,A 34.3587,B 16.8815,C -0.3749,E1 17.0156,E2 414.6361} C_DIS
LIN {X 108.9096,Y 74.1321,Z 160,A 32.4488,B 16.8815,C -0.3701,E1 17.0186,E2 416.5482} C_DIS
LIN {X 111.3993,Y 70.3344,Z 160,A 30.542,B 16.8816,C -0.3677,E1 17.0215,E2 418.4486} C_DIS
LIN {X 113.7552,Y 66.4575,Z 160,A 28.6303,B 16.8817,C -0.3649,E1 17.0242,E2 420.3548} C_DIS
LIN {X 115.8269,Y 62.7774,Z 160,A 26.7419,B 16.8818,C -0.3581,E1 17.0268,E2 422.2511} C_DIS
LIN {X 117.4695,Y 59.6419,Z 160,A 25.3245,B 16.8818,C -0.3586,E1 17.0286,E2 423.6554} C_DIS
LIN {X 119.6711,Y 55.0918,Z 160,A 23.1507,B 16.8819,C -0.3535,E1 17.0312,E2 425.8285} C_DIS
LIN {X 121.0369,Y 52.0228,Z 160,A 21.7064,B 16.882,C -0.3501,E1 17.0328,E2 427.2725} C_DIS
LIN {X 122.2696,Y 49.0554,Z 160,A 20.2764,B 16.8821,C -0.345,E1 17.0343,E2 428.7078} C_DIS
LIN {X 123.4459,Y 46.0151,Z 160,A 18.924,B 16.8821,C -0.3435,E1 17.0356,E2 430.0539} C_DIS
LIN {X 124.5522,Y 42.931,Z 160,A 16.5233,B 16.8829,C -0.3032,E1 17.0379,E2 432.5714} C_DIS
LIN {X 126.5755,Y 36.5399,Z 160,A 14.6203,B 16.8824,C -0.3323,E1 17.0394,E2 434.3584} C_DIS
LIN {X 127.388,Y 33.5962,Z 160,A 13.2931,B 16.8824,C -0.3284,E1 17.0403,E2 435.687} C_DIS
LIN {X 128.7767,Y 27.8002,Z 160,A 10.1667,B 16.8829,C -0.3008,E1 17.0423,E2 438.8799} C_DIS
LIN {X 129.6537,Y 23.3722,Z 160,A 8.7548,B 16.8827,C -0.3155,E1 17.043,E2 440.2289} C_DIS
LIN {X 130.2162,Y 20.0022,Z 160,A 7.3165,B 16.8827,C -0.3129,E1 17.0436,E2 441.6634} C_DIS
LIN {X 130.7275,Y 16.3464,Z 160,A 5.5788,B 16.8829,C -0.303,E1 17.0443,E2 443.419} C_DIS
LIN {X 131.1518,Y 12.4718,Z 160,A 4.0056,B 16.8829,C -0.3025,E1 17.0447,E2 444.9798} C_DIS
LIN {X 131.4733,Y 8.44,Z 160,A 2.2025,B 16.883,C -0.2955,E1 17.0451,E2 446.7905} C_DIS
LIN {X 131.6788,Y 4.1598,Z 160,A 0.3158,B 16.8831,C -0.2889,E1 17.0453,E2 448.6824} C_DIS
LIN {X 131.7447,Y -0.3744,Z 160,A -1.6367,B 16.8832,C -0.2836,E1 17.0453,E2 450.6353} C_DIS
LIN {X 131.6744,Y -4.3178,Z 160,A -3.2077,B 16.8832,C -0.2837,E1 17.0453,E2 452.1914} C_DIS
LIN {X 131.4942,Y -8.1003,Z 160,A -4.8761,B 16.8833,C -0.2779,E1 17.045,E2 453.8646} C_DIS
LIN {X 131.2245,Y -11.6979,Z 160,A -6.5256,B 16.8834,C -0.27,E1 17.0446,E2 455.5259} C_DIS
LIN {X 130.8091,Y -15.662,Z 160,A -8.1163,B 16.8834,C -0.2701,E1 17.0441,E2 457.1018} C_DIS
LIN {X 130.3139,Y -19.3689,Z 160,A -9.9225,B 16.8836,C -0.2583,E1 17.0434,E2 458.932} C_DIS
LIN {X 129.4986,Y -24.2218,Z 160,A -11.8159,B 16.8836,C -0.2611,E1 17.0425,E2 460.7988} C_DIS
LIN {X 127.8844,Y -31.6614,Z 160,A -15.2391,B 16.8838,C -0.2468,E1 17.0404,E2 464.2403} C_DIS
LIN {X 126.2863,Y -37.5277,Z 160,A -17.7165,B 16.8838,C -0.2452,E1 17.0385,E2 466.7015} C_DIS
LIN {X 125.3343,Y -40.5938,Z 160,A -19.24,B 16.8839,C -0.2363,E1 17.0372,E2 468.2422} C_DIS
LIN {X 123.9933,Y -44.5189,Z 160,A -21.1454,B 16.884,C -0.2272,E1 17.0354,E2 470.1624} C_DIS
LIN {X 121.2852,Y -51.4458,Z 160,A -24.1101,B 16.884,C -0.2279,E1 17.0324,E2 473.0995} C_DIS
LIN {X 120.2104,Y -53.9046,Z 160,A -25.2612,B 16.884,C -0.2252,E1 17.0311,E2 474.2502} C_DIS
LIN {X 118.6229,Y -57.3164,Z 160,A -26.9067,B 16.8841,C -0.2202,E1 17.0291,E2 475.8992} C_DIS
LIN {X 117.2986,Y -59.9776,Z 160,A -28.2028,B 16.8841,C -0.2164,E1 17.0275,E2 477.1975} C_DIS
LIN {X 115.0256,Y -64.2339,Z 160,A -30.4033,B 16.8843,C -0.2068,E1 17.0245,E2 479.4133} C_DIS
LIN {X 112.8021,Y -68.062,Z 160,A -32.2489,B 16.8843,C -0.2045,E1 17.0219,E2 481.252} C_DIS
LIN {X 110.644,Y -71.5172,Z 160,A -34.466,B 16.8846,C -0.1832,E1 17.0185,E2 483.525} C_DIS
LIN {X 108.1994,Y -75.1641,Z 160,A -35.885,B 16.8844,C -0.1965,E1 17.0163,E2 484.888} C_DIS
LIN {X 105.8295,Y -78.4661,Z 160,A -38.2115,B 16.8847,C -0.1711,E1 17.0124,E2 487.2838} C_DIS
LIN {X 102.8301,Y -82.3578,Z 160,A -40.3273,B 16.8847,C -0.1666,E1 17.0087,E2 489.4} C_DIS
LIN {X 99.7152,Y -86.1025,Z 160,A -41.9514,B 16.8847,C -0.1797,E1 17.0058,E2 490.9679} C_DIS
LIN {X 97.6632,Y -88.4232,Z 160,A -43.9796,B 16.8849,C -0.1514,E1 17.0019,E2 493.0792} C_DIS
LIN {X 93.5484,Y -92.7655,Z 160,A -45.5861,B 16.8846,C -0.1821,E1 16.999,E2 494.5701} C_DIS
LIN {X 88.4946,Y -97.5984,Z 160,A -48.6354,B 16.8846,C -0.1749,E1 16.9928,E2 497.6244} C_DIS
LIN {X 84.7456,Y -100.8705,Z 160,A -50.9224,B 16.8847,C -0.1658,E1 16.9879,E2 499.9291} C_DIS
LIN {X 82.7716,Y -102.4969,Z 160,A -52.2484,B 16.8848,C -0.1556,E1 16.985,E2 501.2821} C_DIS
LIN {X 79.6799,Y -104.919,Z 160,A -53.8398,B 16.8848,C -0.1565,E1 16.9815,E2 502.8617} C_DIS
LIN {X 76.1413,Y -107.5142,Z 160,A -56.486,B 16.8851,C -0.126,E1 16.9752,E2 505.5981} C_DIS
LIN {X 70.9675,Y -110.9971,Z 160,A -58.3443,B 16.8849,C -0.1521,E1 16.9711,E2 507.3576} C_DIS
LIN {X 67.331,Y -113.24,Z 160,A -60.2384,B 16.8849,C -0.1476,E1 16.9666,E2 509.2581} C_DIS
LIN {X 61.9701,Y -116.2609,Z 160,A -62.8028,B 16.8849,C -0.1472,E1 16.9603,E2 511.8121} C_DIS
LIN {X 59.059,Y -117.7662,Z 160,A -64.8489,B 16.8851,C -0.1226,E1 16.9551,E2 513.934} C_DIS
LIN {X 54.6976,Y -119.8533,Z 160,A -66.3021,B 16.8849,C -0.143,E1 16.9516,E2 515.3116} C_DIS
LIN {X 51.8961,Y -121.0917,Z 160,A -67.6239,B 16.8849,C -0.1416,E1 16.9482,E2 516.6334} C_DIS
LIN {X 48.9571,Y -122.3092,Z 160,A -69.027,B 16.8849,C -0.139,E1 16.9445,E2 518.0402} C_DIS
LIN {X 45.3456,Y -123.6953,Z 160,A -70.8071,B 16.885,C -0.1334,E1 16.9398,E2 519.8338} C_DIS
LIN {X 41.4515,Y -125.0522,Z 160,A -72.4899,B 16.885,C -0.1354,E1 16.9354,E2 521.5048} C_DIS
LIN {X 37.1113,Y -126.4082,Z 160,A -74.572,B 16.885,C -0.1295,E1 16.9298,E2 523.6011} C_DIS
LIN {X 33.7006,Y -127.3601,Z 160,A -76.0251,B 16.885,C -0.1311,E1 16.9259,E2 525.045} C_DIS
LIN {X 29.6555,Y -128.3625,Z 160,A -78.0788,B 16.8851,C -0.121,E1 16.9203,E2 527.1291} C_DIS
LIN {X 24.9394,Y -129.3614,Z 160,A -79.8539,B 16.8851,C -0.1308,E1 16.9155,E2 528.8673} C_DIS
LIN {X 21.438,Y -129.9876,Z 160,A -81.3858,B 16.8851,C -0.1302,E1 16.9113,E2 530.3984} C_DIS
LIN {X 18.4946,Y -130.4388,Z 160,A -82.7715,B 16.8851,C -0.1262,E1 16.9074,E2 531.796} C_DIS
LIN {X 14.3248,Y -130.9625,Z 160,A -84.5768,B 16.8851,C -0.126,E1 16.9024,E2 533.5997} C_DIS
LIN {X 10.7442,Y -131.3051,Z 160,A -86.1454,B 16.8851,C -0.1252,E1 16.8981,E2 535.1698} C_DIS
LIN {X 6.7377,Y -131.5712,Z 160,A -87.88,B 16.8851,C -0.125,E1 16.8932,E2 536.9041} C_DIS
LIN {X 2.8418,Y -131.7145,Z 160,A -89.6773,B 16.8851,C -0.121,E1 16.8882,E2 538.7145} C_DIS
LIN {X 2.8418,Y -131.7145,Z 160,A -89.6773,B 16.8851,C -0.121,E1 16.8882,E2 538.7145} C_DIS
Enddeposition()
LIN {X 0.9299,Y -130.8133,Z 160,A -89.4886,B 14.0889,C 0.1003,E1 14.0903,E2 539.2441} C_DIS
Startdeposition()
$VEL.CP = VEL_PRINT
LIN {X 5.2381,Y -130.7128,Z 160,A -86.8981,B 14.0891,C 0.0793,E1 14.0978,E2 536.5685} C_DIS
LIN {X 9.3243,Y -130.485,Z 160,A -85.2149,B 14.0891,C 0.082,E1 14.1024,E2 534.8975} C_DIS
LIN {X 12.7255,Y -130.1973,Z 160,A -83.6755,B 14.0891,C 0.08,E1 14.1067,E2 533.3518} C_DIS
LIN {X 16.5169,Y -129.7715,Z 160,A -82.0734,B 14.0891,C 0.0812,E1 14.1112,E2 531.7569} C_DIS
LIN {X 19.5827,Y -129.3442,Z 160,A -80.7052,B 14.0891,C 0.0801,E1 14.1149,E2 530.3864} C_DIS
LIN {X 22.4221,Y -128.8831,Z 160,A -79.4373,B 14.0891,C 0.079,E1 14.1184,E2 529.1168} C_DIS
LIN {X 25.3657,Y -128.3367,Z 160,A -77.2684,B 14.0891,C 0.0522,E1 14.1247,E2 526.8429} C_DIS
LIN {X 31.3082,Y -127.0174,Z 160,A -75.5736,B 14.0891,C 0.0794,E1 14.129,E2 525.264} C_DIS
LIN {X 36.9066,Y -125.5033,Z 160,A -72.9133,B 14.0891,C 0.0734,E1 14.1362,E2 522.5872} C_DIS
LIN {X 42.6829,Y -123.6582,Z 160,A -70.3091,B 14.0891,C 0.0721,E1 14.1431,E2 519.9872} C_DIS
LIN {X 45.4169,Y -122.6813,Z 160,A -68.9048,B 14.0891,C 0.0666,E1 14.1468,E2 518.5658} C_DIS
LIN {X 49.2519,Y -121.1921,Z 160,A -67.2228,B 14.0891,C 0.068,E1 14.1511,E2 516.8966} C_DIS
LIN {X 53.035,Y -119.585,Z 160,A -65.6088,B 14.0891,C 0.0713,E1 14.1552,E2 515.3034} C_DIS
LIN {X 56.8935,Y -117.7988,Z 160,A -63.5537,B 14.0891,C 0.0628,E1 14.1605,E2 513.2234} C_DIS
LIN {X 60.5036,Y -115.9851,Z 160,A -61.8122,B 14.0891,C 0.061,E1 14.1648,E2 511.4835} C_DIS
LIN {X 63.1741,Y -114.5544,Z 160,A -60.3817,B 14.0891,C 0.0557,E1 14.1683,E2 510.0393} C_DIS
LIN {X 67.2935,Y -112.1844,Z 160,A -58.3191,B 14.0891,C 0.0529,E1 14.1733,E2 507.9768} C_DIS
LIN {X 70.9743,Y -109.8925,Z 160,A -56.7602,B 14.0891,C 0.0602,E1 14.1769,E2 506.457} C_DIS
LIN {X 74.1848,Y -107.751,Z 160,A -54.7914,B 14.0892,C 0.0485,E1 14.1815,E2 504.4528} C_DIS
LIN {X 77.6635,Y -105.2715,Z 160,A -52.9232,B 14.0892,C 0.0451,E1 14.1857,E2 502.5829} C_DIS
LIN {X 81.1141,Y -102.6366,Z 160,A -51.0765,B 14.0892,C 0.0431,E1 14.1898,E2 500.7408} C_DIS
LIN {X 84.167,Y -100.1477,Z 160,A -49.0144,B 14.0892,C 0.029,E1 14.1943,E2 498.6359} C_DIS
LIN {X 87.0261,Y -97.674,Z 160,A -47.6469,B 14.0892,C 0.0346,E1 14.1971,E2 497.3015} C_DIS
LIN {X 90.3241,Y -94.6318,Z 160,A -45.7121,B 14.0892,C 0.0313,E1 14.201,E2 495.368} C_DIS
LIN {X 93.6106,Y -91.3821,Z 160,A -43.2727,B 14.0892,C 0.0136,E1 14.2059,E2 492.8759} C_DIS
LIN {X 96.6948,Y -88.1125,Z 160,A -41.7582,B 14.0892,C 0.0235,E1 14.2087,E2 491.4141} C_DIS
LIN {X 99.8626,Y -84.5054,Z 160,A -39.1828,B 14.0892,C 0.0035,E1 14.2135,E2 488.7787} C_DIS
LIN {X 102.8566,Y -80.8341,Z 160,A -37.4894,B 14.0892,C 0.0106,E1 14.2163,E2 487.1292} C_DIS
LIN {X 105.9776,Y -76.6967,Z 160,A -35.5155,B 14.0892,C 0.0144,E1 14.2196,E2 485.1882} C_DIS
LIN {X 108.0978,Y -73.6794,Z 160,A -34.0408,B 14.0892,C 0.0148,E1 14.2219,E2 483.7284} C_DIS
LIN {X 110.047,Y -70.7343,Z 160,A -32.2241,B 14.0892,C 0.0022,E1 14.2247,E2 481.8773} C_DIS
LIN {X 112.3367,Y -67.038,Z 160,A -30.3782,B 14.0892,C -0.001,E1 14.2274,E2 480.036} C_DIS
LIN {X 114.5886,Y -63.1124,Z 160,A -28.359,B 14.0892,C -0.0075,E1 14.2302,E2 478.0098} C_DIS
LIN {X 116.5086,Y -59.4884,Z 160,A -26.7663,B 14.0892,C -0.0059,E1 14.2322,E2 476.4392} C_DIS
LIN {X 117.6611,Y -57.1802,Z 160,A -25.2497,B 14.0892,C -0.0214,E1 14.2341,E2 474.8746} C_DIS
LIN {X 119.1217,Y -54.0709,Z 160,A -23.972,B 14.0892,C -0.0183,E1 14.2355,E2 473.6224} C_DIS
LIN {X 123.146,Y -44.1393,Z 160,A -19.4279,B 14.0892,C -0.0267,E1 14.2402,E2 469.0907} C_DIS
LIN {X 124.5293,Y -40.0709,Z 160,A -17.5803,B 14.0892,C -0.031,E1 14.2418,E2 467.2448} C_DIS
LIN {X 125.7395,Y -36.1001,Z 160,A -15.4897,B 14.0892,C -0.0451,E1 14.2435,E2 465.1191} C_DIS
LIN {X 126.6101,Y -32.9184,Z 160,A -14.2637,B 14.0892,C -0.0423,E1 14.2443,E2 463.9177} C_DIS
LIN {X 127.528,Y -29.1511,Z 160,A -12.646,B 14.0892,C -0.0447,E1 14.2454,E2 462.3074} C_DIS
LIN {X 128.4723,Y -24.6593,Z 160,A -10.9838,B 14.0892,C -0.0395,E1 14.2463,E2 460.6843} C_DIS
LIN {X 129.3849,Y -19.3198,Z 160,A -8.2503,B 14.0892,C -0.0581,E1 14.2476,E2 457.9049} C_DIS
LIN {X 129.9021,Y -15.4492,Z 160,A -6.6471,B 14.0892,C -0.0598,E1 14.2481,E2 456.3123} C_DIS
LIN {X 130.3094,Y -11.5309,Z 160,A -4.8485,B 14.0892,C -0.0673,E1 14.2486,E2 454.5029} C_DIS
LIN {X 130.5955,Y -7.6304,Z 160,A -3.1355,B 14.0892,C -0.0724,E1 14.2489,E2 452.7878} C_DIS
LIN {X 130.7807,Y -3.147,Z 160,A -1.1908,B 14.0891,C -0.0777,E1 14.2491,E2 450.8433} C_DIS
LIN {X 130.8159,Y 0.8056,Z 160,A 0.4252,B 14.0891,C -0.0792,E1 14.2491,E2 449.2389} C_DIS
LIN {X 130.7324,Y 4.7365,Z 160,A 2.0859,B 14.0891,C -0.0823,E1 14.2489,E2 447.5836} C_DIS
LIN {X 130.5855,Y 7.794,Z 160,A 3.4318,B 14.0891,C -0.0865,E1 14.2487,E2 446.2355} C_DIS
LIN {X 130.3517,Y 11.0303,Z 160,A 4.8617,B 14.0891,C -0.091,E1 14.2484,E2 444.8029} C_DIS
LIN {X 129.9329,Y 15.1906,Z 160,A 6.5505,B 14.0891,C -0.0919,E1 14.2479,E2 443.129} C_DIS
LIN {X 129.5205,Y 18.376,Z 160,A 8.0978,B 14.0889,C -0.1006,E1 14.2473,E2 441.5634} C_DIS
LIN {X 128.847,Y 22.624,Z 160,A 10.5035,B 14.0888,C -0.1229,E1 14.2462,E2 439.0931} C_DIS
LIN {X 127.9361,Y 27.3062,Z 160,A 12.0643,B 14.0888,C -0.112,E1 14.2453,E2 437.5935} C_DIS
LIN {X 126.9549,Y 31.5602,Z 160,A 13.9599,B 14.0888,C -0.117,E1 14.2441,E2 435.6979} C_DIS
LIN {X 126.1375,Y 34.6817,Z 160,A 15.3439,B 14.0888,C -0.1201,E1 14.2431,E2 434.3159} C_DIS
LIN {X 125.1418,Y 38.1146,Z 160,A 16.7392,B 14.0888,C -0.1191,E1 14.242,E2 432.9393} C_DIS
LIN {X 123.5038,Y 43.1282,Z 160,A 19.0935,B 14.0888,C -0.127,E1 14.2399,E2 430.5776} C_DIS
LIN {X 122.1246,Y 46.8937,Z 160,A 20.8166,B 14.0887,C -0.1308,E1 14.2382,E2 428.8568} C_DIS
LIN {X 120.7713,Y 50.2736,Z 160,A 22.3653,B 14.0887,C -0.1337,E1 14.2366,E2 427.312} C_DIS
LIN {X 119.5084,Y 53.2064,Z 160,A 23.6797,B 14.0887,C -0.1348,E1 14.2351,E2 426.0064} C_DIS
LIN {X 118.0355,Y 56.3979,Z 160,A 25.3042,B 14.0886,C -0.1416,E1 14.2332,E2 424.3704} C_DIS
LIN {X 116.788,Y 58.9397,Z 160,A 26.4029,B 14.0886,C -0.1404,E1 14.2318,E2 423.2875} C_DIS
LIN {X 115.0712,Y 62.2285,Z 160,A 28.2826,B 14.0885,C -0.1527,E1 14.2293,E2 421.3763} C_DIS
LIN {X 113.162,Y 65.6354,Z 160,A 29.9415,B 14.0885,C -0.1554,E1 14.227,E2 419.7221} C_DIS
LIN {X 110.8694,Y 69.4389,Z 160,A 31.9109,B 14.0884,C -0.1611,E1 14.2242,E2 417.7484} C_DIS
LIN {X 108.6505,Y 72.8613,Z 160,A 33.6366,B 14.0884,C -0.1635,E1 14.2215,E2 416.0286} C_DIS
LIN {X 106.5309,Y 75.9266,Z 160,A 35.281,B 14.0884,C -0.1678,E1 14.2189,E2 414.3817} C_DIS
LIN {X 103.7992,Y 79.6203,Z 160,A 37.2621,B 14.0883,C -0.1715,E1 14.2155,E2 412.4029} C_DIS
LIN {X 101.0692,Y 83.0588,Z 160,A 39.1522,B 14.0883,C -0.1749,E1 14.2122,E2 410.5155} C_DIS
LIN {X 98.3145,Y 86.302,Z 160,A 40.9228,B 14.0883,C -0.1761,E1 14.209,E2 408.7548} C_DIS
LIN {X 93.9449,Y 91.0383,Z 160,A 43.8183,B 14.0881,C -0.1843,E1 14.2035,E2 405.8492} C_DIS
LIN {X 90.8234,Y 94.153,Z 160,A 45.709,B 14.0881,C -0.187,E1 14.1997,E2 403.9624} C_DIS
LIN {X 87.6904,Y 97.0778,Z 160,A 47.5598,B 14.0881,C -0.1899,E1 14.1959,E2 402.1139} C_DIS
LIN {X 84.4782,Y 99.8858,Z 160,A 49.3756,B 14.0881,C -0.1918,E1 14.1921,E2 400.3035} C_DIS
LIN {X 79.6363,Y 103.7869,Z 160,A 52.1578,B 14.0879,C -0.1984,E1 14.186,E2 397.5135} C_DIS
LIN {X 76.3877,Y 106.2011,Z 160,A 53.958,B 14.0879,C -0.2023,E1 14.1819,E2 395.7095} C_DIS
LIN {X 72.7474,Y 108.7266,Z 160,A 55.8626,B 14.0879,C -0.2043,E1 14.1775,E2 393.8085} C_DIS
LIN {X 68.9453,Y 111.1765,Z 160,A 57.8528,B 14.0878,C -0.2076,E1 14.1728,E2 391.8168} C_DIS
LIN {X 65.0731,Y 113.4866,Z 160,A 59.7851,B 14.0878,C -0.2091,E1 14.1682,E2 389.8892} C_DIS
LIN {X 61.7719,Y 115.3165,Z 160,A 61.4454,B 14.0878,C -0.2116,E1 14.1641,E2 388.2278} C_DIS
LIN {X 58.4285,Y 117.0453,Z 160,A 63.0901,B 14.0878,C -0.2136,E1 14.16,E2 386.5833} C_DIS
LIN {X 54.593,Y 118.8816,Z 160,A 64.9143,B 14.0877,C -0.2147,E1 14.1554,E2 384.7635} C_DIS
LIN {X 50.6448,Y 120.6163,Z 160,A 66.6934,B 14.0877,C -0.2135,E1 14.1508,E2 382.9972} C_DIS
LIN {X 47.5651,Y 121.8636,Z 160,A 68.0055,B 14.0877,C -0.2108,E1 14.1475,E2 381.7018} C_DIS
LIN {X 44.6687,Y 122.9551,Z 160,A 69.6257,B 14.0877,C -0.2199,E1 14.1432,E2 380.0507} C_DIS
LIN {X 40.3706,Y 124.4336,Z 160,A 71.5157,B 14.0877,C -0.2186,E1 14.1382,E2 378.1727} C_DIS
LIN {X 37.237,Y 125.4066,Z 160,A 72.7966,B 14.0877,C -0.2152,E1 14.1348,E2 376.9102} C_DIS
LIN {X 33.1479,Y 126.5493,Z 160,A 74.8979,B 14.0876,C -0.2236,E1 14.1291,E2 374.7809} C_DIS
LIN {X 29.5168,Y 127.4445,Z 160,A 76.4298,B 14.0876,C -0.2215,E1 14.125,E2 373.2617} C_DIS
LIN {X 26.1392,Y 128.1793,Z 160,A 78.3336,B 14.0874,C -0.2336,E1 14.1196,E2 371.3126} C_DIS
LIN {X 22.3253,Y 128.9004,Z 160,A 79.7319,B 14.0875,C -0.2256,E1 14.1159,E2 369.9502} C_DIS
LIN {X 19.0652,Y 129.422,Z 160,A 81.1194,B 14.0875,C -0.2244,E1 14.1121,E2 368.5699} C_DIS
LIN {X 15.511,Y 129.8947,Z 160,A 82.6986,B 14.0875,C -0.2251,E1 14.1077,E2 366.9902} C_DIS
LIN {X 11.245,Y 130.3336,Z 160,A 84.4584,B 14.0875,C -0.2221,E1 14.1028,E2 365.2448} C_DIS
LIN {X 8.2044,Y 130.5602,Z 160,A 85.8919,B 14.0875,C -0.2251,E1 14.0988,E2 363.8004} C_DIS
LIN {X 4.0448,Y 130.7558,Z 160,A 87.7607,B 14.0875,C -0.2264,E1 14.0936,E2 361.9272} C_DIS
LIN {X -0.1122,Y 130.8191,Z 160,A 89.6089,B 14.0875,C -0.2271,E1 14.0884,E2 360.0767} C_DIS
LIN {X -4.5077,Y 130.7413,Z 160,A 91.534,B 14.0875,C -0.2267,E1 14.083,E2 358.1526} C_DIS
LIN {X -8.3267,Y 130.5526,Z 160,A 93.2248,B 14.0875,C -0.2267,E1 14.0783,E2 356.4608} C_DIS
LIN {X -12.9734,Y 130.1735,Z 160,A 95.2172,B 14.0875,C -0.2247,E1 14.0728,E2 354.4754} C_DIS
LIN {X -16.8607,Y 129.7264,Z 160,A 97.0345,B 14.0875,C -0.2268,E1 14.0677,E2 352.647} C_DIS
LIN {X -20.4482,Y 129.2102,Z 160,A 98.9908,B 14.0874,C -0.2362,E1 14.0622,E2 350.6485} C_DIS
LIN {X -24.7682,Y 128.4515,Z 160,A 100.6045,B 14.0875,C -0.2264,E1 14.0579,E2 349.0722} C_DIS
LIN {X -28.5811,Y 127.6582,Z 160,A 102.7443,B 14.0873,C -0.2372,E1 14.052,E2 346.8829} C_DIS
LIN {X -33.4107,Y 126.4792,Z 160,A 104.201,B 14.0877,C -0.2154,E1 14.0482,E2 345.5121} C_DIS
LIN {X -36.741,Y 125.5518,Z 160,A 105.7824,B 14.0877,C -0.2159,E1 14.044,E2 343.9241} C_DIS
LIN {X -39.982,Y 124.5577,Z 160,A 107.6974,B 14.0875,C -0.2263,E1 14.0387,E2 341.96} C_DIS
LIN {X -43.6919,Y 123.3072,Z 160,A 109.1534,B 14.0877,C -0.2173,E1 14.035,E2 340.5358} C_DIS
LIN {X -47.0385,Y 122.0683,Z 160,A 110.6071,B 14.0877,C -0.2126,E1 14.0312,E2 339.0962} C_DIS
LIN {X -50.685,Y 120.5995,Z 160,A 112.6636,B 14.0877,C -0.2196,E1 14.0258,E2 337.0021} C_DIS
LIN {X -53.9826,Y 119.1612,Z 160,A 114.0005,B 14.0877,C -0.211,E1 14.0225,E2 335.6946} C_DIS
LIN {X -57.5916,Y 117.4581,Z 160,A 115.655,B 14.0878,C -0.2061,E1 14.0184,E2 334.0525} C_DIS
LIN {X -61.1097,Y 115.6669,Z 160,A 117.9342,B 14.0876,C -0.2184,E1 14.0126,E2 331.7108} C_DIS
LIN {X -65.1479,Y 113.4439,Z 160,A 119.5414,B 14.0878,C -0.2042,E1 14.0088,E2 330.1538} C_DIS
LIN {X -68.7772,Y 111.2811,Z 160,A 121.1899,B 14.088,C -0.1958,E1 14.0049,E2 328.5306} C_DIS
LIN {X -72.0971,Y 109.159,Z 160,A 123.0836,B 14.088,C -0.1973,E1 14.0004,E2 326.6192} C_DIS
LIN {X -75.3127,Y 106.9656,Z 160,A 125.0787,B 14.0879,C -0.202,E1 13.9958,E2 324.5921} C_DIS
LIN {X -78.1195,Y 104.9332,Z 160,A 126.3502,B 14.088,C -0.1926,E1 13.993,E2 323.351} C_DIS
LIN {X -81.6993,Y 102.1711,Z 160,A 128.2273,B 14.088,C -0.1861,E1 13.9889,E2 321.488} C_DIS
LIN {X -84.2333,Y 100.0921,Z 160,A 129.7631,B 14.088,C -0.1859,E1 13.9856,E2 319.9422} C_DIS
LIN {X -87.4617,Y 97.2838,Z 160,A 131.6578,B 14.0881,C -0.1826,E1 13.9816,E2 318.0472} C_DIS
LIN {X -90.4759,Y 94.4868,Z 160,A 133.4252,B 14.0881,C -0.1779,E1 13.9781,E2 316.2858} C_DIS
LIN {X -92.5464,Y 92.4604,Z 160,A 134.6517,B 14.0882,C -0.174,E1 13.9756,E2 315.0658} C_DIS
LIN {X -95.0573,Y 89.8764,Z 160,A 136.3418,B 14.0882,C -0.1734,E1 13.9724,E2 313.3645} C_DIS
LIN {X -97.7393,Y 86.953,Z 160,A 138.1621,B 14.0882,C -0.1716,E1 13.9689,E2 311.5366} C_DIS
LIN {X -100.6254,Y 83.5955,Z 160,A 140.1104,B 14.0883,C -0.1673,E1 13.9654,E2 309.5896} C_DIS
LIN {X -103.3767,Y 80.1678,Z 160,A 142.5419,B 14.0883,C -0.1759,E1 13.9612,E2 307.1012} C_DIS
LIN {X -106.2725,Y 76.2879,Z 160,A 144.1809,B 14.0884,C -0.158,E1 13.9586,E2 305.5212} C_DIS
LIN {X -109.1603,Y 72.095,Z 160,A 146.4135,B 14.0884,C -0.1525,E1 13.9551,E2 303.2911} C_DIS
LIN {X -111.4973,Y 68.4251,Z 160,A 148.2425,B 14.0886,C -0.1456,E1 13.9524,E2 301.4733} C_DIS
LIN {X -113.5562,Y 64.951,Z 160,A 150.1124,B 14.0886,C -0.1435,E1 13.9497,E2 299.594} C_DIS
LIN {X -116.1166,Y 60.2532,Z 160,A 152.4197,B 14.0886,C -0.1363,E1 13.9467,E2 297.2938} C_DIS
LIN {X -118.0185,Y 56.4335,Z 160,A 154.1381,B 14.0887,C -0.1273,E1 13.9446,E2 295.5952} C_DIS
LIN {X -119.1807,Y 53.9389,Z 160,A 155.5957,B 14.0887,C -0.1304,E1 13.9429,E2 294.1098} C_DIS
LIN {X -120.6182,Y 50.6402,Z 160,A 156.9137,B 14.0887,C -0.1195,E1 13.9415,E2 292.8238} C_DIS
LIN {X -121.8027,Y 47.7217,Z 160,A 158.2833,B 14.0888,C -0.1153,E1 13.9401,E2 291.4572} C_DIS
LIN {X -122.9776,Y 44.6063,Z 160,A 159.9899,B 14.0888,C -0.1175,E1 13.9384,E2 289.7235} C_DIS
LIN {X -123.9299,Y 41.8912,Z 160,A 161.3296,B 14.0888,C -0.1159,E1 13.9372,E2 288.3761} C_DIS
LIN {X -125.0423,Y 38.4398,Z 160,A 162.8499,B 14.0888,C -0.1096,E1 13.9359,E2 286.8658} C_DIS
LIN {X -126.1807,Y 34.5273,Z 160,A 164.7068,B 14.0889,C -0.1062,E1 13.9345,E2 285.0028} C_DIS
LIN {X -127.1363,Y 30.8151,Z 160,A 166.3811,B 14.0889,C -0.1012,E1 13.9334,E2 283.3311} C_DIS
LIN {X -127.7859,Y 28.002,Z 160,A 167.5659,B 14.0889,C -0.0954,E1 13.9326,E2 282.1572} C_DIS
LIN {X -128.3845,Y 25.1182,Z 160,A 168.806,B 14.089,C -0.0903,E1 13.932,E2 280.9246} C_DIS
LIN {X -128.984,Y 21.8272,Z 160,A 170.4848,B 14.089,C -0.0914,E1 13.9311,E2 279.2226} C_DIS
LIN {X -129.587,Y 17.9104,Z 160,A 172.2676,B 14.089,C -0.0875,E1 13.9304,E2 277.4365} C_DIS
LIN {X -130.0174,Y 14.4543,Z 160,A 173.7738,B 14.089,C -0.0824,E1 13.9299,E2 275.9344} C_DIS
LIN {X -130.3056,Y 11.576,Z 160,A 174.9742,B 14.089,C -0.0769,E1 13.9296,E2 274.7434} C_DIS
LIN {X -130.6861,Y 5.9023,Z 160,A 177.4002,B 14.0891,C -0.0678,E1 13.9292,E2 272.3281} C_DIS
LIN {X -130.8032,Y 1.9559,Z 160,A 179.3485,B 14.0891,C -0.0682,E1 13.9291,E2 270.3561} C_DIS
LIN {X -130.6417,Y -6.785,Z 160,A -176.9276,B 14.0891,C -0.054,E1 13.9294,E2 266.6492} C_DIS
LIN {X -130.1014,Y -13.6733,Z 160,A -173.803,B 14.0892,C -0.0475,E1 13.9301,E2 263.5166} C_DIS
LIN {X -129.4921,Y -18.5747,Z 160,A -171.6231,B 14.0892,C -0.0415,E1 13.9309,E2 261.3372} C_DIS
LIN {X -128.8714,Y -22.4872,Z 160,A -169.8734,B 14.0892,C -0.0368,E1 13.9317,E2 259.5877} C_DIS
LIN {X -128.2481,Y -25.8012,Z 160,A -168.2758,B 14.0892,C -0.0356,E1 13.9326,E2 257.9775} C_DIS
LIN {X -127.2528,Y -30.3319,Z 160,A -166.3314,B 14.0892,C -0.0275,E1 13.9338,E2 256.0456} C_DIS
LIN {X -126.5298,Y -33.2208,Z 160,A -165.0616,B 14.0892,C -0.0229,E1 13.9346,E2 254.7811} C_DIS
LIN {X -125.5918,Y -36.6046,Z 160,A -163.4484,B 14.0892,C -0.0204,E1 13.9359,E2 253.1606} C_DIS
LIN {X -124.5906,Y -39.8792,Z 160,A -161.9285,B 14.0892,C -0.0167,E1 13.9371,E2 251.6398} C_DIS
LIN {X -123.2802,Y -43.767,Z 160,A -160.0266,B 14.0892,C -0.0144,E1 13.9389,E2 249.7274} C_DIS
LIN {X -122.1504,Y -46.8273,Z 160,A -158.4475,B 14.0892,C -0.0144,E1 13.9405,E2 248.1318} C_DIS
LIN {X -120.2026,Y -51.6194,Z 160,A -156.4142,B 14.0892,C -0.0022,E1 13.9426,E2 246.128} C_DIS
LIN {X -118.9911,Y -54.3561,Z 160,A -154.3923,B 14.0892,C -0.0173,E1 13.9451,E2 244.0229} C_DIS
LIN {X -116.7764,Y -58.9624,Z 160,A -152.7422,B 14.0892,C 0.0041,E1 13.9471,E2 242.4447} C_DIS
LIN {X -114.9859,Y -62.3855,Z 160,A -150.9853,B 14.0892,C 0.0067,E1 13.9494,E2 240.6816} C_DIS
LIN {X -113.1826,Y -65.5998,Z 160,A -149.2517,B 14.0892,C 0.0077,E1 13.9518,E2 238.9351} C_DIS
LIN {X -110.2129,Y -70.4752,Z 160,A -146.2055,B 14.0892,C -0.0006,E1 13.9565,E2 235.8256} C_DIS
LIN {X -107.1474,Y -75.0548,Z 160,A -144.3887,B 14.0892,C 0.021,E1 13.9592,E2 234.0818} C_DIS
LIN {X -104.5543,Y -78.6262,Z 160,A -142.4992,B 14.0892,C 0.0267,E1 13.9623,E2 232.1988} C_DIS
LIN {X -102.5647,Y -81.2048,Z 160,A -140.9805,B 14.0892,C 0.0275,E1 13.965,E2 230.6701} C_DIS
LIN {X -99.6661,Y -84.7366,Z 160,A -139.1883,B 14.0892,C 0.0374,E1 13.9681,E2 228.9038} C_DIS
LIN {X -97.8521,Y -86.8254,Z 160,A -137.4843,B 14.0892,C 0.0269,E1 13.9714,E2 227.1419} C_DIS
LIN {X -95.3207,Y -89.5971,Z 160,A -136.1531,B 14.0892,C 0.0387,E1 13.9739,E2 225.8489} C_DIS
LIN {X -92.4076,Y -92.5988,Z 160,A -134.27,B 14.0892,C 0.0411,E1 13.9776,E2 223.9607} C_DIS
LIN {X -88.2025,Y -96.6131,Z 160,A -131.6958,B 14.0892,C 0.0453,E1 13.9828,E2 221.3844} C_DIS
LIN {X -85.3248,Y -99.163,Z 160,A -129.3114,B 14.0892,C 0.0294,E1 13.9881,E2 218.9166} C_DIS
LIN {X -80.8166,Y -102.8703,Z 160,A -127.4529,B 14.0892,C 0.0529,E1 13.9919,E2 217.143} C_DIS
LIN {X -77.1878,Y -105.6209,Z 160,A -125.4631,B 14.0892,C 0.0564,E1 13.9964,E2 215.1544} C_DIS
LIN {X -73.8369,Y -107.9898,Z 160,A -123.643,B 14.0892,C 0.0586,E1 14.0006,E2 213.332} C_DIS
LIN {X -70.6114,Y -110.1257,Z 160,A -122.2086,B 14.0892,C 0.0683,E1 14.0038,E2 211.929} C_DIS
LIN {X -67.8948,Y -111.8212,Z 160,A -120.5275,B 14.0892,C 0.0627,E1 14.0079,E2 210.215} C_DIS
LIN {X -63.9863,Y -114.1026,Z 160,A -118.5961,B 14.0892,C 0.0668,E1 14.0126,E2 208.29} C_DIS
LIN {X -60.0936,Y -116.2004,Z 160,A -116.5239,B 14.0892,C 0.0655,E1 14.0177,E2 206.2019} C_DIS
LIN {X -56.4367,Y -118.017,Z 160,A -114.926,B 14.0892,C 0.0729,E1 14.0217,E2 204.6269} C_DIS
LIN {X -53.6119,Y -119.327,Z 160,A -113.5344,B 14.0892,C 0.0737,E1 14.0252,E2 203.232} C_DIS
LIN {X -50.5469,Y -120.6572,Z 160,A -112.1386,B 14.0891,C 0.0771,E1 14.0288,E2 201.8443} C_DIS
LIN {X -47.6621,Y -121.8259,Z 160,A -110.6368,B 14.0891,C 0.0745,E1 14.0327,E2 200.326} C_DIS
LIN {X -44.3933,Y -123.0544,Z 160,A -109.1961,B 14.0891,C 0.0784,E1 14.0365,E2 198.8958} C_DIS
LIN {X -41.4892,Y -124.0638,Z 160,A -107.7979,B 14.0891,C 0.0781,E1 14.0402,E2 197.4913} C_DIS
LIN {X -36.1925,Y -125.7124,Z 160,A -105.2853,B 14.0891,C 0.0775,E1 14.0469,E2 194.9685} C_DIS
LIN {X -32.5596,Y -126.7012,Z 160,A -103.6312,B 14.0891,C 0.0784,E1 14.0514,E2 193.3136} C_DIS
LIN {X -25.9244,Y -128.223,Z 160,A -100.6885,B 14.0891,C 0.081,E1 14.0594,E2 190.3749} C_DIS
LIN {X -21.7203,Y -129.0018,Z 160,A -98.8338,B 14.0891,C 0.0822,E1 14.0645,E2 188.5219} C_DIS
LIN {X -18.3014,Y -129.5311,Z 160,A -97.2665,B 14.0891,C 0.0812,E1 14.0689,E2 186.9479} C_DIS
LIN {X -14.5731,Y -130.0046,Z 160,A -95.5853,B 14.0891,C 0.0805,E1 14.0735,E2 185.262} C_DIS
LIN {X -10.7021,Y -130.3794,Z 160,A -93.9148,B 14.0891,C 0.0816,E1 14.0782,E2 183.5948} C_DIS
LIN {X -6.9676,Y -130.6325,Z 160,A -92.2508,B 14.0891,C 0.081,E1 14.0828,E2 181.9271} C_DIS
LIN {X -2.5313,Y -130.7937,Z 160,A -90.3476,B 14.0891,C 0.082,E1 14.0881,E2 180.0279} C_DIS
LIN {X 0.9299,Y -130.8133,Z 160,A -89.4861,B 14.0889,C 0.1009,E1 14.0903,E2 179.244} C_DIS
Enddeposition()
LIN {X 0.9299,Y -130.8133,Z 160,A -89.4861,B 14.0889,C 0.1009,E1 14.0903,E2 179.244} C_DIS
Startdeposition()
$VEL.CP = VEL_PRINT
LIN {X -0.0054,Y -129.8937,Z 160,A -90.1077,B 14.0891,C 0.0982,E1 14.0888,E2 179.8544} C_DIS
LIN {X -4.3139,Y -129.822,Z 160,A -91.8362,B 14.0891,C 0.0934,E1 14.084,E2 181.5634} C_DIS
LIN {X -7.4919,Y -129.6764,Z 160,A -93.2845,B 14.0891,C 0.0947,E1 14.08,E2 183.0176} C_DIS
LIN {X -11.1496,Y -129.4124,Z 160,A -94.9405,B 14.0891,C 0.0956,E1 14.0753,E2 184.6788} C_DIS
LIN {X -15.4372,Y -128.971,Z 160,A -96.849,B 14.0891,C 0.0955,E1 14.07,E2 186.5887} C_DIS
LIN {X -18.5918,Y -128.5543,Z 160,A -98.1921,B 14.0891,C 0.0934,E1 14.0663,E2 187.9252} C_DIS
LIN {X -22.2,Y -127.9822,Z 160,A -99.8252,B 14.0891,C 0.0934,E1 14.0618,E2 189.5614} C_DIS
LIN {X -25.8426,Y -127.2948,Z 160,A -101.541,B 14.0891,C 0.095,E1 14.0571,E2 191.2869} C_DIS
LIN {X -29.585,Y -126.4791,Z 160,A -103.1339,B 14.0891,C 0.0915,E1 14.0528,E2 192.869} C_DIS
LIN {X -32.6654,Y -125.7191,Z 160,A -104.5383,B 14.0891,C 0.0908,E1 14.049,E2 194.2741} C_DIS
LIN {X -35.7271,Y -124.8837,Z 160,A -105.9441,B 14.0891,C 0.09,E1 14.0452,E2 195.6809} C_DIS
LIN {X -38.7964,Y -123.9645,Z 160,A -107.3626,B 14.0892,C 0.0891,E1 14.0414,E2 197.1002} C_DIS
LIN {X -41.8214,Y -122.9769,Z 160,A -109.0007,B 14.0892,C 0.0944,E1 14.037,E2 198.7659} C_DIS
LIN {X -45.6975,Y -121.5874,Z 160,A -110.6517,B 14.0892,C 0.0883,E1 14.0327,E2 200.3975} C_DIS
LIN {X -49.2713,Y -120.1859,Z 160,A -112.2978,B 14.0892,C 0.0853,E1 14.0285,E2 202.0382} C_DIS
LIN {X -52.2012,Y -118.9423,Z 160,A -113.7025,B 14.0892,C 0.0839,E1 14.0249,E2 203.4429} C_DIS
LIN {X -55.036,Y -117.6567,Z 160,A -115.1975,B 14.0892,C 0.0856,E1 14.021,E2 204.9521} C_DIS
LIN {X -58.4093,Y -116.019,Z 160,A -116.7352,B 14.0892,C 0.0805,E1 14.0172,E2 206.4761} C_DIS
LIN {X -61.2361,Y -114.5533,Z 160,A -118.0739,B 14.0892,C 0.0769,E1 14.0139,E2 207.8068} C_DIS
LIN {X -64.0249,Y -113.0186,Z 160,A -119.5653,B 14.0892,C 0.0774,E1 14.0103,E2 209.3082} C_DIS
LIN {X -66.7749,Y -111.4156,Z 160,A -120.9806,B 14.0892,C 0.0758,E1 14.0069,E2 210.7246} C_DIS
LIN {X -69.6356,Y -109.6506,Z 160,A -122.5814,B 14.0892,C 0.0768,E1 14.0031,E2 212.3389} C_DIS
LIN {X -73.106,Y -107.3679,Z 160,A -124.3154,B 14.0893,C 0.0713,E1 13.9991,E2 214.0609} C_DIS
LIN {X -75.7151,Y -105.5438,Z 160,A -125.7253,B 14.0893,C 0.0692,E1 13.9958,E2 215.4711} C_DIS
LIN {X -78.2784,Y -103.6567,Z 160,A -127.0824,B 14.0893,C 0.0656,E1 13.9928,E2 216.8222} C_DIS
LIN {X -81.2015,Y -101.3839,Z 160,A -128.8304,B 14.0893,C 0.0658,E1 13.989,E2 218.5831} C_DIS
LIN {X -84.2507,Y -98.8639,Z 160,A -130.6437,B 14.0893,C 0.0644,E1 13.9851,E2 220.4036} C_DIS
LIN {X -87.2122,Y -96.2614,Z 160,A -132.3879,B 14.0893,C 0.0613,E1 13.9814,E2 222.1477} C_DIS
LIN {X -90.1422,Y -93.5238,Z 160,A -134.2194,B 14.0893,C 0.0594,E1 13.9777,E2 223.9857} C_DIS
LIN {X -93.3594,Y -90.312,Z 160,A -136.1778,B 14.0893,C 0.0541,E1 13.9739,E2 225.9375} C_DIS
LIN {X -96.3059,Y -87.1632,Z 160,A -137.8395,B 14.0894,C 0.0438,E1 13.9708,E2 227.5703} C_DIS
LIN {X -98.2099,Y -85.0127,Z 160,A -139.3363,B 14.0894,C 0.0471,E1 13.968,E2 229.0931} C_DIS
LIN {X -100.5537,Y -82.2264,Z 160,A -141.0034,B 14.0894,C 0.0451,E1 13.965,E2 230.7663} C_DIS
LIN {X -103.2328,Y -78.8368,Z 160,A -142.8652,B 14.0894,C 0.0396,E1 13.9618,E2 232.6217} C_DIS
LIN {X -105.2714,Y -76.0934,Z 160,A -144.3476,B 14.0894,C 0.0355,E1 13.9594,E2 234.1003} C_DIS
LIN {X -107.1303,Y -73.453,Z 160,A -145.7807,B 14.0894,C 0.0323,E1 13.9571,E2 235.5333} C_DIS
LIN {X -108.8898,Y -70.8185,Z 160,A -147.1881,B 14.0894,C 0.0292,E1 13.9549,E2 236.9409} C_DIS
LIN {X -110.9594,Y -67.5306,Z 160,A -148.9528,B 14.0894,C 0.0262,E1 13.9523,E2 238.7102} C_DIS
LIN {X -112.7881,Y -64.4289,Z 160,A -150.5234,B 14.0894,C 0.0218,E1 13.9501,E2 240.2776} C_DIS
LIN {X -114.5552,Y -61.2326,Z 160,A -152.1596,B 14.0894,C 0.0183,E1 13.9479,E2 241.9154} C_DIS
LIN {X -116.5396,Y -57.3606,Z 160,A -154.0886,B 14.0894,C 0.0135,E1 13.9455,E2 243.8438} C_DIS
LIN {X -118.0997,Y -54.0779,Z 160,A -155.7118,B 14.0894,C 0.0097,E1 13.9436,E2 245.4679} C_DIS
LIN {X -119.3865,Y -51.1739,Z 160,A -157.1166,B 14.0894,C 0.0061,E1 13.942,E2 246.8719} C_DIS
LIN {X -120.7744,Y -47.8113,Z 160,A -158.9339,B 14.0894,C 0.0071,E1 13.9401,E2 248.7123} C_DIS
LIN {X -122.0662,Y -44.4041,Z 160,A -160.5088,B 14.0894,C 0.0018,E1 13.9386,E2 250.282} C_DIS
LIN {X -123.3347,Y -40.7482,Z 160,A -162.0928,B 14.0894,C -0.0061,E1 13.9372,E2 251.8501} C_DIS
LIN {X -124.3005,Y -37.6995,Z 160,A -163.5173,B 14.0894,C -0.0097,E1 13.936,E2 253.2748} C_DIS
LIN {X -125.187,Y -34.6425,Z 160,A -164.9353,B 14.0894,C -0.0133,E1 13.9349,E2 254.693} C_DIS
LIN {X -125.9991,Y -31.5623,Z 160,A -166.354,B 14.0894,C -0.017,E1 13.9339,E2 256.1119} C_DIS
LIN {X -126.7408,Y -28.4396,Z 160,A -167.7826,B 14.0894,C -0.0208,E1 13.933,E2 257.5404} C_DIS
LIN {X -127.3065,Y -25.785,Z 160,A -169.0535,B 14.0894,C -0.0224,E1 13.9323,E2 258.8185} C_DIS
LIN {X -127.9819,Y -22.202,Z 160,A -170.6008,B 14.0894,C -0.0287,E1 13.9315,E2 260.3572} C_DIS
LIN {X -128.487,Y -19.0628,Z 160,A -172.055,B 14.0894,C -0.0315,E1 13.9309,E2 261.8158} C_DIS
LIN {X -128.9723,Y -15.4267,Z 160,A -173.7388,B 14.0894,C -0.0346,E1 13.9303,E2 263.5052} C_DIS
LIN {X -129.4157,Y -11.1107,Z 160,A -175.6141,B 14.0894,C -0.0413,E1 13.9298,E2 265.3739} C_DIS
LIN {X -129.6477,Y -7.9572,Z 160,A -176.955,B 14.0894,C -0.0468,E1 13.9295,E2 266.707} C_DIS
LIN {X -129.821,Y -4.3445,Z 160,A -178.8101,B 14.0894,C -0.0451,E1 13.9293,E2 268.5902} C_DIS
LIN {X -129.8946,Y -0.0859,Z 160,A 179.476,B 14.0894,C -0.0548,E1 13.9293,E2 270.283} C_DIS
LIN {X -129.8581,Y 3.0164,Z 160,A 178.1606,B 14.0894,C -0.0602,E1 13.9293,E2 271.5906} C_DIS
LIN {X -129.7856,Y 5.2538,Z 160,A 177.0513,B 14.0894,C -0.0602,E1 13.9295,E2 272.7127} C_DIS
LIN {X -129.5719,Y 9.1146,Z 160,A 175.3477,B 14.0894,C -0.0653,E1 13.9297,E2 274.414} C_DIS
LIN {X -129.2193,Y 13.2161,Z 160,A 173.3479,B 14.0894,C -0.0662,E1 13.9303,E2 276.4326} C_DIS
LIN {X -128.711,Y 17.4834,Z 160,A 171.639,B 14.0893,C -0.0765,E1 13.9309,E2 278.1179} C_DIS
LIN {X -128.3168,Y 20.1666,Z 160,A 170.3383,B 14.0893,C -0.0774,E1 13.9314,E2 279.429} C_DIS
LIN {X -127.7854,Y 23.3,Z 160,A 168.9808,B 14.0893,C -0.0827,E1 13.9321,E2 280.7797} C_DIS
LIN {X -127.1021,Y 26.7819,Z 160,A 167.4545,B 14.0893,C -0.0883,E1 13.9329,E2 282.2996} C_DIS
LIN {X -126.4847,Y 29.5607,Z 160,A 166.1302,B 14.0892,C -0.0903,E1 13.9337,E2 283.6302} C_DIS
LIN {X -125.723,Y 32.65,Z 160,A 164.7092,B 14.0892,C -0.0939,E1 13.9347,E2 285.0515} C_DIS
LIN {X -124.8859,Y 35.7192,Z 160,A 163.2891,B 14.0892,C -0.0976,E1 13.9358,E2 286.4717} C_DIS
LIN {X -123.974,Y 38.7665,Z 160,A 161.8695,B 14.0892,C -0.1012,E1 13.9369,E2 287.8914} C_DIS
LIN {X -122.8265,Y 42.2553,Z 160,A 160.1264,B 14.0892,C -0.1028,E1 13.9385,E2 289.6464} C_DIS
LIN {X -121.3549,Y 46.3182,Z 160,A 158.3038,B 14.0891,C -0.1103,E1 13.9402,E2 291.4572} C_DIS
LIN {X -120.1803,Y 49.2852,Z 160,A 156.8774,B 14.0891,C -0.1138,E1 13.9417,E2 292.8839} C_DIS
LIN {X -118.9377,Y 52.2118,Z 160,A 155.4594,B 14.0891,C -0.1173,E1 13.9433,E2 294.3019} C_DIS
LIN {X -117.4229,Y 55.5323,Z 160,A 153.8447,B 14.089,C -0.1217,E1 13.9452,E2 295.9151} C_DIS
LIN {X -116.0278,Y 58.392,Z 160,A 152.4293,B 14.089,C -0.1252,E1 13.9469,E2 297.33} C_DIS
LIN {X -114.565,Y 61.2143,Z 160,A 151.0839,B 14.0889,C -0.1304,E1 13.9487,E2 298.6672} C_DIS
LIN {X -113.0815,Y 63.9132,Z 160,A 149.6117,B 14.0889,C -0.1312,E1 13.9507,E2 300.1507} C_DIS
LIN {X -111.1653,Y 67.1901,Z 160,A 147.8185,B 14.0889,C -0.1326,E1 13.9533,E2 301.9553} C_DIS
LIN {X -109.1357,Y 70.4398,Z 160,A 146.2423,B 14.0888,C -0.1398,E1 13.9556,E2 303.5164} C_DIS
LIN {X -107.1068,Y 73.4872,Z 160,A 144.4918,B 14.0888,C -0.1405,E1 13.9584,E2 305.2803} C_DIS
LIN {X -104.5423,Y 77.0921,Z 160,A 142.5581,B 14.0888,C -0.1458,E1 13.9615,E2 307.2096} C_DIS
LIN {X -102.2479,Y 80.1101,Z 160,A 140.8438,B 14.0888,C -0.1488,E1 13.9645,E2 308.9266} C_DIS
LIN {X -99.7476,Y 83.2033,Z 160,A 139.0547,B 14.0887,C -0.152,E1 13.9676,E2 310.7176} C_DIS
LIN {X -96.9352,Y 86.4631,Z 160,A 137.2102,B 14.0887,C -0.1578,E1 13.971,E2 312.5535} C_DIS
LIN {X -94.2426,Y 89.3906,Z 160,A 135.3845,B 14.0886,C -0.16,E1 13.9745,E2 314.3852} C_DIS
LIN {X -91.2777,Y 92.4162,Z 160,A 133.4845,B 14.0886,C -0.1632,E1 13.9782,E2 316.2867} C_DIS
LIN {X -88.4051,Y 95.1672,Z 160,A 131.7315,B 14.0886,C -0.167,E1 13.9818,E2 318.0374} C_DIS
LIN {X -85.4493,Y 97.8297,Z 160,A 130.0279,B 14.0885,C -0.1719,E1 13.9853,E2 319.7333} C_DIS
LIN {X -82.3973,Y 100.414,Z 160,A 128.1825,B 14.0885,C -0.1733,E1 13.9893,E2 321.586} C_DIS
LIN {X -79.283,Y 102.8911,Z 160,A 126.4669,B 14.0884,C -0.1777,E1 13.9931,E2 323.2951} C_DIS
LIN {X -76.0765,Y 105.2836,Z 160,A 124.7498,B 14.0884,C -0.1822,E1 13.9969,E2 325.0049} C_DIS
LIN {X -73.4811,Y 107.111,Z 160,A 123.3434,B 14.0883,C -0.1845,E1 14.0001,E2 326.4105} C_DIS
LIN {X -70.8412,Y 108.875,Z 160,A 121.8426,B 14.0883,C -0.1843,E1 14.0037,E2 327.9213} C_DIS
LIN {X -67.1827,Y 111.1698,Z 160,A 120.013,B 14.0883,C -0.1894,E1 14.008,E2 329.7404} C_DIS
LIN {X -64.3917,Y 112.8093,Z 160,A 118.5814,B 14.0883,C -0.1916,E1 14.0114,E2 331.171} C_DIS
LIN {X -61.5734,Y 114.3721,Z 160,A 117.0972,B 14.0882,C -0.1921,E1 14.0151,E2 332.6609} C_DIS
LIN {X -58.8079,Y 115.8161,Z 160,A 115.7663,B 14.0882,C -0.1953,E1 14.0184,E2 333.9853} C_DIS
LIN {X -55.9578,Y 117.2196,Z 160,A 114.2866,B 14.0882,C -0.1952,E1 14.0221,E2 335.4726} C_DIS
LIN {X -52.6459,Y 118.7448,Z 160,A 112.7391,B 14.0882,C -0.1989,E1 14.026,E2 337.0116} C_DIS
Enddeposition()
END
